(* CODESYS project oaksmodbuslibrary.library
   Title: oaksModbusLibrary
   Version: 1.1
   Placeholder: oaksModbusLibrary
   Company: Oaks AB

Project tree, tasks and I/O mapping:
  libraries: OaksLibrary, 1.1 (OaksAB); Tc2_BA, 3.3.9.0 (Beckhoff Automation GmbH); Tc2_ModbusSrv, 3.3.2.0 (Beckhoff Automation GmbH); Tc2_Standard, 3.3.3.0 (Beckhoff Automation GmbH); Tc2_System, 3.4.24.0 (Beckhoff Automation GmbH); Tc2_Utilities, 3.3.47.0 (Beckhoff Automation GmbH); Tc3_BA, 1.1.5.0 (Beckhoff Automation GmbH); Tc3_BA_Common, 2.1.4.0 (Beckhoff Automation GmbH); Tc3_Module, 3.3.21.0 (Beckhoff Automation GmbH)
  oaksModbusLibrary/
    [obsolete]/
      function block fbRCCC3DOCS [ST]
      function block fbSioxDamper [ST]
      function block fbWriteHoldingDoubleControlled [ST]
      function fHyst [ST]
    Belimo/
      Spjällställdon/
        function block fbBelimoLHVD3MOD [ST]
        function block fbBelimoUK24MOD [ST]
    Bitzer/
      function block fbBitzerSEi1 [ST]
    Calectro/
      function block fbCalair [ST]
      function block fbCalectroIoMb02 [ST]
    Daikin/
      function block fbDaikinRTDNET [ST]
    Danfoss/
      function block fbDanfossDGS_HFC [ST]
      function block fbDanfossEKE347 [ST]
    Datahantering/
      function F_INT_TO_WORD [ST]
      function F_WORD_TO_INT [ST]
      function block FB_SETPOINT_INT_MODBUS [ST]
      function block FB_SETPOINT_REAL_MODBUS [ST]
      function block fbDoubleControlledModbusHolding [ST]
      function block fbHoldingRWReadBackEEPROM_BOOL [ST]
      function block fbHoldingRWReadBackEEPROM_REAL [ST]
      function block fbReadGeneralModbusReg [ST]
      function block fbReadWriteCoilRegBool [ST]
      function block fbReadWriteHoldingReg [ST]
      function block fbReadWriteHoldingRegReal [ST]
      function fWordToReal [ST]
    DUTs/
      data type E_Modbus_Functions_Read
      data type ST_ModbusConfig
      data type ST_ModbusData
      data type ST_ModbusResultRegister
      data type ST_ModbusTCP
      data type U_WORD_INT
    EBM Papst/
      function block fbEbmPapst [ST]
    EcoGuard/
      function block fbEcocomTemperature [ST]
    Ej Testat/
    Elvaco/
      CME3100/
        Givare/
          function block fbElvacoTemperature [ST]
          function block fbElvacoTemperatureCo2 [ST]
          function block fbElvacoTemperatureHumidity [ST]
        Mätare/
          function block fbElvacoElectricMeter [ST]
          function block fbElvacoElectricMeterEnergy [ST]
          function block fbElvacoEnergyMeter [ST]
          function block fbElvacoWaterMeter [ST]
        function block fbElvacoGeneral [ST]
    Eveco/
      function block fbEveco [ST]: mSpeedEnableCheck
    Fidelix/
      FXIO (IO-kort)/
        Givarblock/
          function block fbFxIO_Sensor [ST]: mGT, mRaw
        Modulblock/
          function block fbFxIO_AI8 [ST]: mAI
          function block fbFxIO_AO8 [ST]
          function block fbFxIO_Combi36 [ST]
          function block fbFxIO_DI16 [ST]
          function block fbFxIO_DO8 [ST]
    Fläktwoods/
      Spjällställdon/
        function block fbFlaktwoods227PMMB [ST]
        function block fbFlaktwoods227VMMB [ST]
    Frico/
      function block fbFricoSirE [ST]: mBHyst
      function block fbFricoSirEOvride [ST]: mBHyst
    Grundfil/
      function block fbGrundfil [ST]
    Grundfos/
      function block fbGrundfosCIM [ST]
      function block fbGrundfosModbusMagna [ST]
    Gruner/
      Givare/
        function block fbGrunerGTVMDD3MB [ST]
      Spjällställdon/
        function block fbGruner227CMXXMB [ST]
    IMI hydronic/
      function block fbImiBrainCubeConnect [ST]
    Iv produkt/
      function block fbIvClimatixEnvistarIndication [ST]
      function block fbIvClimatixEnvistarOperationLevel [CFC]: mCommunicationAlarm, mIpadressString, mSpeedChoice
      function block fbIvSaphirOperationLevel [CFC]: mCommunicationAlarm, mIpadressString, mSpeedChoice
    IVT/
      function block fbIvtRego5200BorVarde [ST]
    Metz/
      DUT/
        data type E_MetzAIsensorConfig
        data type ST_MetzAI8config
        data type ST_MetzAI8Sensor
      Givare/
        function block fbMetzMR_AI8GeneralSensor [ST]
        function block fbMetzMR_AI8TempSensor [ST]
      function block fbMetzMR_AI8 [ST]: config
      function block fbMetzMR_AOP4 [ST]: mAnalogToRaw, mAnalogToRawFallback, mRawToAnalog
      function block fbMetzMR_DI10 [ST]
      function block fbMetzMR_DI4 [ST]
      function block fbMetzMR_DO4 [ST]: mAnalogToRaw, mAnalogToRawFallback, mRawToAnalog
      function block fbMetzMR_MULTI [ST]: config, mAnalogIn, mAnalogOut, mAnalogToRaw, mAnalogToRawFallback, mDigitalIn, mDigitalOut, mRawToAnalog
    Mitsubishi/
      function block fbMitsubishiATA_ATW [ST]
      function block fbMitsubishiHydroBox [ST]
    Nicotra Gebhardt/
      function block fbNicotraGebhardtRLM [ST]
    Produal/
      Givare/
        function block fbProdualHdhmCo2 [ST]
        function block fbProdualHdhmPirCo2 [ST]
        function block fbProdualHdhmTempCo2 [ST]
        function block fbProdualKLH [ST]
        function block fbProdualPEL2500Mx [ST]
      ProximaRIO/
        function block fbProximaCULH_RIO [ST]: mADConfig, mINConfig
        function block fbProximaRIO_Sensor [ST]: mDataIn
        data type ST_ProximaCULH_IO_Config
      Regulatorer/
        HLS44/
          function block fbProdualHLS44 [ST]
          function block fbProdualHLS44_IO [ST]
        function block fbProdualHdhmCo2Override [ST]
        function block fbProdualHdhmCo2PirOverride [ST]
    Regin/
      Givare/
        function block fbCthrc [ST]
        function block fbCtrc [ST]
      Regio midi/
        function block fbReginRCC [ST]
        function block fbReginRCC_CO2 [ST]
        function block fbReginRCC_Handst_Spjall [ST]
        function block fbReginRCC_Handst_Spjall_Co2 [ST]
    Schneider/
      function block fbAltivarATV600 [ST]
    Server-block/
      RTU/
        function block fbMbRtuSlaveCoilRegBool [ST]
        function block fbMbRtuSlaveHoldingRegInt [ST]
        function block fbMbRtuSlaveHoldingRegReal [ST]
        function block fbMbRtuSlaveHoldingRegUInt [ST]
        function block fbMbRtuSlaveStatusRegBool [ST]
      function block fbMbSlaveRegBool [ST]
      function block fbMbSlaveRegInt [ST]
      function block fbMbSlaveRegReal [ST]
      function block fbMbSlaveRegUInt [ST]
    Siemens/
      Spjäll/
        function block fbSiemensGDB1811EMO [ST]
    Siox/
      Via modul/
        function block fbSioxDamperDUOdirect [ST]
        function block fbSioxDamperUNOdirect [ST]
        function block fbSioxSxAcura [ST]
      Via SX-Access/
        function block fbSioxDamperDUO [ST]
        function block fbSioxDamperUNO [ST]
      function block fbSioxSxAcess [ST]
    Swegon/
      function block fbSwegonGoldCdOperationLevel [CFC]: mCommunicationAlarm, mIpadressString, mSpeedChoice
      function block fbSwegonGoldIndication [ST]
      function block fbSwegonGoldOperationLevel [CFC]: mCommunicationAlarm, mIpadressString, mSpeedChoice
      function block fbSwegonReact [ST]: mFlodesBalansering, mFlodesKompensering1, mFlodesKompensering10, mFlodesKompensering11, mFlodesKompensering12, mFlodesKompensering13, mFlodesKompensering14, mFlodesKompensering15, mFlodesKompensering2, mFlodesKompensering3, mFlodesKompensering4, mFlodesKompensering5, mFlodesKompensering6, mFlodesKompensering7, mFlodesKompensering8, mFlodesKompensering9, mOperationMode
      function block fbSwegonReactPx [ST]
      function block fbSwegonWiseMasterSlave [ST]
    Vacon/
      function block fbVaconFO_1 [ST]
    Wilo/
      function block fbWiloCif_If [ST]
    Xylem/
      function block fbXylemEcocircXLplus [ST]
      function block fbXylemHydrovarHVL [ST]
  ClassDiagram
  global variables GVL_ModbusRtuSlave
  global variables ModbusServer
*)

// oaksModbusLibrary/DUTs/E_Modbus_Functions_Read
{attribute 'qualified_only'}
{attribute 'strict'}
TYPE E_Modbus_Functions_Read :
(
	ReadCoils 			:= 1,
	ReadInputStatus 	:= 2,
	ReadHoldingRegister	:= 3,
	ReadInputRegister	:= 4
);
END_TYPE

// oaksModbusLibrary/DUTs/ST_ModbusConfig
TYPE ST_ModbusConfig :
STRUCT
	bEnable 		: BOOL; // IF TRUE, the slave is present and will be read from terminal. If FALSE no read are done and no update of values
	eMBFunction		: E_Modbus_Functions_Read; //MODBUS FUNCTION to use.
	nUnitId			: BYTE; // The MOdbus DeviceId of slave (1..247)
	nQuantity		: WORD :=1; // Quantity of registers or coils to be read out from slave (1..125 for holding/input registers, 1..2000 for coils)
	nMBAddr			: WORD; // The startaddress of the register or coil to be read out from slave
	tTimeBetwRead 	: TIME :=T#500MS; // Time before readout of the slave
END_STRUCT
END_TYPE

// oaksModbusLibrary/DUTs/ST_ModbusData
TYPE ST_ModbusData :
STRUCT
	aModbusData			: ARRAY [1..1000] OF WORD;
	aModbusGoodRead		: ARRAY [1..1000] OF BOOL;
	aModbusAddress		: ARRAY [1..1000] OF UINT;
	aModbusTimestamp	: ARRAY [1..1000] OF DT;
END_STRUCT
END_TYPE

// oaksModbusLibrary/DUTs/ST_ModbusResultRegister
TYPE ST_ModbusResultRegister :
STRUCT
	bEnable 		: BOOL; // IF TRUE, the slave is present and will be read from terminal. If false no read are done and no update of values
	eMBFunction		: E_Modbus_Functions_Read; //MODBUS FUNCTION that have been used
	nUnitId			: BYTE; // The MOdbus DeviceId of slave (1..247)
	nQuantity		: WORD; // Quantity of registers or coils to be read out from slave (1..125 for holding/input registers, 1..2000 for coils)
	nMBAddr			: WORD; // The startaddress of the register or coil to be read out from slave
	aRegisterArray	: ARRAY [1..125] OF WORD; // The telegram maximum length is 125 values of WORD.
	bReadSuccessful	: BOOL; // If the last read out from slave is without error then this value is TRUE, else FALSE
	DTLastRead		: TIMESTRUCT; // The date and time for the last reafout from slave (the values in aRegisterarray is from this date)
	stModbusError	: ST_ModbusErrorDiagnostics; // Error diagnostics from the last readout
	
END_STRUCT
END_TYPE

// oaksModbusLibrary/DUTs/ST_ModbusTCP
TYPE ST_ModbusTCP :
STRUCT
	sIPAddr : STRING := ''; //Ip-adress
	nTCPPort : UINT; //Modbus-TCP port
	iModbusLoop : INT :=1; //Modbusslinga
END_STRUCT
END_TYPE

// oaksModbusLibrary/DUTs/U_WORD_INT
TYPE U_WORD_INT :
UNION
	nWord	: WORD;
	nINT	: INT;
END_UNION
END_TYPE

// oaksModbusLibrary/Metz/DUT/E_MetzAIsensorConfig
{attribute 'qualified_only'}
{attribute 'strict'}
{attribute 'to_string'}
TYPE E_MetzAIsensorConfig :
(
Sensor_PT100 := 0,
Sensor_PT500 := 1,
Sensor_PT1000 := 2,
Sensor_NI1000_TK5000 := 3,
Sensor_NI1000_TK6180 := 4,
Sensor_BALCO_500 := 5,
Sensor_KTY81_110 := 6,
Sensor_KTY81_210 := 7,
Sensor_NTC_1k8 := 8,
Sensor_NTC_5k := 9,
Sensor_NTC_10k := 10,
Sensor_NTC_20k := 11,
Sensor_LM235 := 12,
Sensor_NTC_10k_CAREL := 13
);
END_TYPE

// oaksModbusLibrary/Metz/DUT/ST_MetzAI8config
TYPE ST_MetzAI8config :
STRUCT
	bResistance : BOOL :=FALSE; //0=0-10v, 1=Resistans
	sensorType : E_MetzAIsensorConfig := 2;  
END_STRUCT
END_TYPE

// oaksModbusLibrary/Metz/DUT/ST_MetzAI8Sensor
TYPE ST_MetzAI8Sensor :
STRUCT
	rRawValue : REAL := 0; //Rå-värde från IO-modul 
	bComError : BOOL := FALSE; //Kommunikationsfel från IO-modul
	sSensorConfig : STRING := ' '; 
END_STRUCT
END_TYPE

// oaksModbusLibrary/Produal/ProximaRIO/ST_ProximaCULH_IO_Config
TYPE ST_ProximaCULH_IO_Config :
STRUCT
	nInType 	: BYTE;
	nInRType	: BYTE; //0=Ohm, 1=DI
	nInDelay	: BYTE;
	
	nOutType	: BYTE; //0=0..10V, 1=PWM
	iOutPW		: INT;

	bError		: BOOL;	
END_STRUCT
END_TYPE

// GVL_ModbusRtuSlave
{attribute 'qualified_only'}
VAR_GLOBAL PERSISTENT
mb_Input    :  ARRAY [0..999] OF WORD;
mb_Output 	:  ARRAY [0..999] OF WORD;
mb_Memory	:  ARRAY [0..999] OF WORD;
END_VAR

// ModbusServer
{attribute 'qualified_only'}
VAR_GLOBAL
	mb_HoldingRegs 	:    ARRAY [0..999] OF WORD;
	mb_Coils	 	:    ARRAY [0..999] OF BOOL;
END_VAR

// oaksModbusLibrary/[obsolete]/fbRCCC3DOCS
//OAKS AB
//2020-03-17
//Funktionsblock för modbus-TCP, Regin RCC-C3DOCS rumsreglator (Endast som börvärdesomställare) bör ej användas för rumsstyrning.
// Specifikt för krokslätts fabriker.
{attribute 'obsolete' := 'Använd ersättningsblock. Detta block vidareutvecklas ej.'}
FUNCTION_BLOCK fbRCCC3DOCS
VAR_INPUT
	sIPAddr : STRING := ''; 
	nTCPPort : UINT := 502;
	nUnitID : UINT :=1;
	iModbusLoop : INT :=1; //Modbusslinga
	iMode : INT; //Driftläge 0=Off 1=Unoccupied, 2=Stand-by, 3=Occupied, 4=Bypass 
	bBlockDisplay : BOOL := TRUE;  //Blockering display
	iSetViewDisp : INT;//Visningsläge i display 0=Ärvärde, 1=Värmebörvärde, 2=Kylbörvärde, 3=Medelvärdet av värme och kylbörvärdet, 4=Endast börvärdesjusteringen, se modbuslista Adr 51
	iSetvalDisp : INT; //Visning av börvärde vid börvärdesjustering, se modbuslista Adr 52
	iBypassTime : INT; //Bypass-tid (min)
	rActSetpoint : REAL; //Aktuellt börvärde
	rActMaxSetpoint : REAL; //Max börvärdeförskjutning
	rActMinSetpoint : REAL; //Min börvärdeförskjutning
END_VAR

VAR_OUTPUT
	PV AT %M* : REAL;//Rumstemperatur~wp:[unit]°C[format]0.0[trendoptions]i:300
	PV1 AT %M* : INT;//Koldioxid~wp:[unit]ppm[format]0[trendoptions]i:300
	PV2 AT %M* : REAL;//Aktuell börvärdesförskjutning~wp:[unit]°C[format]0.0[trendoptions]i:300
	PV7 AT %M* : INT;//Modbus-ID~wp:[format]0
	PV8 AT %M* : INT;//Driftläge~wp:[format]0[trendoptions]i:300
	PV9 AT %M* : REAL;//Max lokal börvärdesförskutning~wp:[unit]°C[format]0.0[trendoptions]i:300
	PV10 AT %M* : REAL;//Min lokal börvärdesförskutning~wp:[unit]°C[format]0.0[trendoptions]i:300
	
	FAULT AT %M* : BOOL;//Kommunikationsfel~wp:
END_VAR

VAR
	//General
	offset : INT;
	rTemp : REAL;
	iTemp : INT;
	wTemp : WORD;
	bSekvensFlagga : BOOL;
	bBlockDisplayRead :  BOOL;
	
	//Read Coils
	FB_MBReadCoils_BlockDisp: FB_MBReadCoils;
	FB_MBWriteCoils_BlockDisp: FB_MBWriteCoils;
	
	//Read input registers
	FB_MBReadInputRegs_wArrInput1: FB_MBReadInputRegs;
	wArrInputRegs1 : ARRAY [1..12] OF WORD; //Input register function 4
		
	FB_MBReadInputRegs_wCo2: FB_MBReadInputRegs;		
	wCO2 : WORD; //Input register function 4
	
	//Read Holding	
	FB_MBReadRegs_Mode : FB_MBReadRegs;
	wModeRead : WORD; //Aktuellt driftläge 0=Off 1=Unoccupied, 2=Stand-by, 3=Occupied, 4=Bypass 

	FB_MBReadRegs_wArrHolding1 : FB_MBReadRegs;
	wArrHolding1 : ARRAY [51..60] OF WORD; //Holding
	wViewDispRead : WORD; //Visningsläge display, se modbus-lista
	wSetValDispRead : WORD; //Visningsläge börvärde, se modbus-lista
	wBypassTimeRead : WORD; //Tid i by-pass läge
		
	FB_MBReadRegs_wArrHolding2: FB_MBReadRegs;
	wArrHolding2 : ARRAY [61..80] OF WORD; //Holding
	wActSetpointRead : WORD; //Grundbörvärde kyla
	wActMaxSetpointRead : WORD; //Max förskjutning lokalt börvärde
	wActMinSetpointRead : WORD; //Min förskjutning lokalt börvärde
	wActOffsetRead : WORD; //Börvärdesjustering
	
	//Write Holding
	FB_MBWriteSingleReg_Mode : FB_MBWriteSingleReg;
	FB_MBWriteSingleReg_SetView : FB_MBWriteSingleReg;
	FB_MBWriteSingleReg_SetDisp : FB_MBWriteSingleReg;
	FB_MBWriteSingleReg_Bypasstime : FB_MBWriteSingleReg;
	FB_MBWriteSingleReg_Setpoint : FB_MBWriteSingleReg;
	FB_MBWriteSingleReg_MaxSetpoint : FB_MBWriteSingleReg;
	FB_MBWriteSingleReg_MinSetpoint : FB_MBWriteSingleReg;
	
	//Kommunikationsfel
	fbKommTof : tof; 
	fbKommTon : ton;
	
	FB_MBReadRegs_ArrHolding1: INT;
	bError: INT;
END_VAR

//General
	offset := -1;
//Sekvens	
	bSekvensFlagga := oaksGVL.aBModbusSekvens[iModbusLoop] = UINT_TO_INT(nUnitID);
//Modbus-ID
	PV7 :=  UINT_TO_INT(nUnitID);
///////////////		
//READ
///////////////			

//Read/Write Coils
	
	//Block display read
	FB_MBReadCoils_BlockDisp(
		sIPAddr:= sIpAddr, 
		nTCPPort:= INT_TO_UINT(nTCPPort), 
		nUnitID:= INT_TO_BYTE(nUnitID), 
		nQuantity:=1, 
		nMBAddr:= 21 + offset, 
		cbLength:= SIZEOF(bBlockDisplayRead), 
		pDestAddr:= ADR(bBlockDisplayRead), 
		bExecute:= bSekvensFlagga, 
		tTimeout:= T#3S, 
		bBusy=> , 
		bError=> , 
		nErrId=> , 
		cbRead=> );
				
		IF bBlockDisplay <> bBlockDisplayRead AND bSekvensFlagga THEN
			FB_MBWriteCoils_BlockDisp.bExecute := TRUE;
		ELSE
			FB_MBWriteCoils_BlockDisp.bExecute := FALSE;
		END_IF

	//Block display write	
	FB_MBWriteCoils_BlockDisp(
		sIPAddr:= sIpAddr, 
		nTCPPort:= INT_TO_UINT(nTCPPort), 
		nUnitID:= INT_TO_BYTE(nUnitID), 
		nQuantity:= 1, 
		nMBAddr:= 21 + offset, 
		cbLength:= SIZEOF(bBlockDisplay), 
		pSrcAddr:= ADR(bBlockDisplay), 
		bExecute:= , 
		tTimeout:= , 
		bBusy=> , 
		bError=> , 
		nErrId=> );	

		
//Read input registers function 4		

	//Read Array1
	FB_MBReadInputRegs_wArrInput1(
		sIPAddr:= sIpAddr, 
		nTCPPort:= INT_TO_UINT(nTCPPort), 
		nUnitID:= INT_TO_BYTE(nUnitID), 
		nQuantity:= 12, 
		nMBAddr:= 1 + offset, 
		cbLength:= SIZEOF(wArrInputRegs1), 
		pDestAddr:= ADR(wArrInputRegs1), 
		bExecute:= bSekvensFlagga, 
		tTimeout:= T#3S, 
		bBusy=> , 
		bError=> , 
		nErrId=> , 
		cbRead=> );
	
		//Values
		//wArrInputRegs1[1]; //1
		//wArrInputRegs1[2]; //2
		//wArrInputRegs1[3]; //3
		//wArrInputRegs1[4]; //4
		//wArrInputRegs1[5]; //5
		//wArrInputRegs1[6]; //6
		//wArrInputRegs1[7]); //7
		//wArrInputRegs1[8]; //8
		//wArrInputRegs1[9]; //9
		//wArrInputRegs1[10]; //10
		iTemp := WORD_TO_INT(wArrInputRegs1[11]); //11
		rTemp := INT_TO_REAL(iTemp); 
		PV := rTemp /10;
		//wArrInputRegs1[12]; //12
	
	//Read CO2		
	FB_MBReadInputRegs_wCo2(
		sIPAddr:= sIpAddr, 
		nTCPPort:= INT_TO_UINT(nTCPPort), 
		nUnitID:= INT_TO_BYTE(nUnitID), 
		nQuantity:= 1, 
		nMBAddr:= 32 + offset, 
		cbLength:= SIZEOF(wCO2), 
		pDestAddr:= ADR(wCO2), 
		bExecute:= bSekvensFlagga, 
		tTimeout:= T#3S, 
		bBusy=> , 
		bError=> , 
		nErrId=> , 
		cbRead=> );
	
		PV1 := WORD_TO_INT(wCO2); //32

//Read Holding registers function 3		

	//Read Mode
	FB_MBReadRegs_Mode(
		sIPAddr:= sIpAddr, 
		nTCPPort:= INT_TO_UINT(nTCPPort), 
		nUnitID:= INT_TO_BYTE(nUnitID), 
		nQuantity:= 1, 
		nMBAddr:= 14+offset, 
		cbLength:= SIZEOF(wModeRead), 
		pDestAddr:= ADR(wModeRead), 
		bExecute:= bSekvensFlagga, 
		tTimeout:= T#3S, 
		bBusy=> , 
		bError=> , 
		nErrId=> , 
		cbRead=> );

		PV8 := WORD_TO_INT(wModeRead);
		
	//Read Array1	
	FB_MBReadRegs_wArrHolding1(
		sIPAddr:= sIpAddr, 
		nTCPPort:= INT_TO_UINT(nTCPPort), 
		nUnitID:= INT_TO_BYTE(nUnitID), 
		nQuantity:= 10, 
		nMBAddr:= 51+offset, 
		cbLength:= SIZEOF(wArrHolding1), 
		pDestAddr:= ADR(wArrHolding1), 
		bExecute:= bSekvensFlagga, 
		tTimeout:= T#3S, 
		bBusy=> , 
		bError=> , 
		nErrId=> , 
		cbRead=> );
		
		//Values
		wViewDispRead := wArrHolding1[51]; //51
		wSetValDispRead := wArrHolding1[52]; //52
		//wArrHolding1[53]; //53
		//wArrHolding1[54]; //54
		//wArrHolding1[55]; //55
		wBypassTimeRead := wArrHolding1[56]; //56
		//wArrHolding1[57]; //57
		//wArrHolding1[58]; //58
		//wArrHolding1[59]; //59
		//wArrHolding1[60]; //60

	//Read Array2	
	FB_MBReadRegs_wArrHolding2(
		sIPAddr:= sIpAddr, 
		nTCPPort:= INT_TO_UINT(nTCPPort), 
		nUnitID:= INT_TO_BYTE(nUnitID), 
		nQuantity:= 20, 
		nMBAddr:= 61+offset, 
		cbLength:= SIZEOF(wArrHolding2), 
		pDestAddr:= ADR(wArrHolding2), 
		bExecute:= bSekvensFlagga, 
		tTimeout:= T#3S, 
		bBusy=> , 
		bError=> , 
		nErrId=> , 
		cbRead=> );
		
		//Values
		//wArrHolding2[61]; //61
		//wArrHolding2[62]; //62
		//wArrHolding2[63]; //63
		//wArrHolding2[64]; //64
		//wArrHolding2[65]; //65
		//wArrHolding2[66]; //66
		//wArrHolding2[67]; //67
		//wArrHolding2[68]; //68
		wActSetpointRead := (wArrHolding2[69]); //69
		//wArrHolding2[70]; //70
		//wArrHolding2[71]; //71
		//wArrHolding2[72]; //72
		//wArrHolding2[73]; //73
		
		wActMaxSetpointRead := (wArrHolding2[74]); //74
		iTemp := WORD_TO_INT(wActMaxSetpointRead);		
		PV9 := iTemp / 10;
		
		wActMinSetpointRead := (wArrHolding2[75]); //75
		iTemp := WORD_TO_INT(wActMinSetpointRead);	
		PV10 := iTemp /10;
		
		wActOffsetRead := (wArrHolding2[76]); //76
		iTemp := WORD_TO_INT(wActOffsetRead);
		PV2 := iTemp / 10;
		
		//wArrHolding2[77]; //77
		//wArrHolding2[78]; //78
		//wArrHolding2[79]; //79
		//wArrHolding2[80]; //80

//Write Holding registers

	//Write mode
	wTemp := INT_TO_WORD(iMode);
	
	IF (wModeRead) <> wTemp AND bSekvensFlagga THEN
		FB_MBWriteSingleReg_Mode.bExecute := TRUE;
	ELSE
		FB_MBWriteSingleReg_Mode.bExecute := FALSE;
	END_IF

	FB_MBWriteSingleReg_Mode(
		sIPAddr:= sIpAddr , 
		nTCPPort:= INT_TO_UINT(nTCPPort), 
		nUnitID:= INT_TO_BYTE(nUnitID), 
		nMBAddr:= 14 + offset, 
		nValue:= wTemp, 
		bExecute:= , 
		tTimeout:= T#5S , 
		bBusy=> , 
		bError=> , 
		nErrId=> );
	
	//Write Viewmode
	wTemp := INT_TO_WORD(iSetViewDisp);
	
	IF wViewDispRead <> wTemp AND bSekvensFlagga THEN
		FB_MBWriteSingleReg_SetView.bExecute := TRUE;
	ELSE
		FB_MBWriteSingleReg_SetView.bExecute := FALSE;
	END_IF

	FB_MBWriteSingleReg_SetView(
		sIPAddr:= sIpAddr , 
		nTCPPort:= INT_TO_UINT(nTCPPort), 
		nUnitID:= INT_TO_BYTE(nUnitID), 
		nMBAddr:= 51 + offset, 
		nValue:= wTemp, 
		bExecute:= , 
		tTimeout:= T#5S , 
		bBusy=> , 
		bError=> , 
		nErrId=> );
		
	//Write DisplaySetpoint Mode
	wTemp := INT_TO_WORD(iSetvalDisp);
	
	IF wSetValDispRead <> wTemp AND bSekvensFlagga THEN
		FB_MBWriteSingleReg_SetDisp.bExecute := TRUE;
	ELSE
		FB_MBWriteSingleReg_SetDisp.bExecute := FALSE;
	END_IF

	FB_MBWriteSingleReg_SetDisp(
		sIPAddr:= sIpAddr , 
		nTCPPort:= INT_TO_UINT(nTCPPort), 
		nUnitID:= INT_TO_BYTE(nUnitID), 
		nMBAddr:= 52 + offset, 
		nValue:= wTemp, 
		bExecute:= , 
		tTimeout:= T#5S , 
		bBusy=> , 
		bError=> , 
		nErrId=> );

	//Write Bypass-time
	wTemp := INT_TO_WORD(iBypassTime);
	
	IF wBypassTimeRead <> wTemp AND bSekvensFlagga THEN
		FB_MBWriteSingleReg_Bypasstime.bExecute := TRUE;
	ELSE
		FB_MBWriteSingleReg_Bypasstime.bExecute := FALSE;
	END_IF

	FB_MBWriteSingleReg_Bypasstime(
		sIPAddr:= sIpAddr , 
		nTCPPort:= INT_TO_UINT(nTCPPort), 
		nUnitID:= INT_TO_BYTE(nUnitID), 
		nMBAddr:= 56 + offset, 
		nValue:= wTemp, 
		bExecute:= , 
		tTimeout:= T#5S , 
		bBusy=> , 
		bError=> , 
		nErrId=> );

	//Setpoint
	iTemp := REAL_TO_INT(rActSetpoint * 10);
	wTemp := INT_TO_WORD(iTemp);
	
	IF wActSetpointRead <> wTemp AND bSekvensFlagga THEN
		FB_MBWriteSingleReg_Setpoint.bExecute := TRUE;
	ELSE
		FB_MBWriteSingleReg_Setpoint.bExecute := FALSE;
	END_IF

	FB_MBWriteSingleReg_Setpoint(
		sIPAddr:= sIpAddr , 
		nTCPPort:= INT_TO_UINT(nTCPPort), 
		nUnitID:= INT_TO_BYTE(nUnitID), 
		nMBAddr:= 69 + offset, 
		nValue:= wTemp, 
		bExecute:= , 
		tTimeout:= T#5S , 
		bBusy=> , 
		bError=> , 
		nErrId=> );
	
	//Max Setpoint
	iTemp := REAL_TO_INT(rActMaxSetpoint * 10);
	wTemp := INT_TO_WORD(iTemp);
	
	IF wActMaxSetpointRead <> wTemp AND bSekvensFlagga THEN
		FB_MBWriteSingleReg_MaxSetpoint.bExecute := TRUE;
	ELSE
		FB_MBWriteSingleReg_MaxSetpoint.bExecute := FALSE;
	END_IF

	FB_MBWriteSingleReg_MaxSetpoint(
		sIPAddr:= sIpAddr , 
		nTCPPort:= INT_TO_UINT(nTCPPort), 
		nUnitID:= INT_TO_BYTE(nUnitID), 
		nMBAddr:= 74 + offset, 
		nValue:= wTemp, 
		bExecute:= , 
		tTimeout:= T#5S , 
		bBusy=> , 
		bError=> , 
		nErrId=> );	
		
	//Min Setpoint
	iTemp := REAL_TO_INT(rActMinSetpoint * 10);
	wTemp := INT_TO_WORD(iTemp);
	
	IF wActMinSetpointRead <> wTemp AND bSekvensFlagga THEN
		FB_MBWriteSingleReg_MinSetpoint.bExecute := TRUE;
	ELSE
		FB_MBWriteSingleReg_MinSetpoint.bExecute := FALSE;
	END_IF

	FB_MBWriteSingleReg_MinSetpoint(
		sIPAddr:= sIpAddr , 
		nTCPPort:= INT_TO_UINT(nTCPPort), 
		nUnitID:= INT_TO_BYTE(nUnitID), 
		nMBAddr:= 75 + offset, 
		nValue:= wTemp, 
		bExecute:= , 
		tTimeout:= T#5S , 
		bBusy=> , 
		bError=> , 
		nErrId=> );	

//Communication error
	fbKommTof(IN:=FB_MBReadCoils_BlockDisp.bError OR
	FB_MBWriteCoils_BlockDisp.bError OR		
	FB_MBReadInputRegs_wArrInput1.bError OR
	FB_MBReadInputRegs_wCo2.bError OR	
	FB_MBReadRegs_Mode.bError OR
	FB_MBReadRegs_wArrHolding1.bError OR
	FB_MBReadRegs_wArrHolding2.bError OR
	FB_MBWriteSingleReg_Mode.bError OR
	FB_MBWriteSingleReg_SetView.bError OR
	FB_MBWriteSingleReg_SetDisp.bError OR
	FB_MBWriteSingleReg_Bypasstime.bError OR
	FB_MBWriteSingleReg_Setpoint.bError OR
	FB_MBWriteSingleReg_MaxSetpoint.bError OR
	FB_MBWriteSingleReg_MinSetpoint.bError,
	PT:=T#20S , Q=> , ET=> );
	fbKommTon(IN:=fbKommTof.Q , PT:=T#20M , Q=> , ET=> );
	FAULT :=fbKommTon.Q;

//Write busy	
	oaksgvl.aBModbusBusyFlagga[iModbusLoop,nUnitID] := FB_MBReadCoils_BlockDisp.bBusy OR
	FB_MBWriteCoils_BlockDisp.bBusy OR		
	FB_MBReadInputRegs_wArrInput1.bBusy OR
	FB_MBReadInputRegs_wCo2.bBusy OR	
	FB_MBReadRegs_Mode.bBusy OR
	FB_MBReadRegs_wArrHolding1.bBusy OR
	FB_MBReadRegs_wArrHolding2.bBusy OR
	FB_MBWriteSingleReg_Mode.bBusy OR
	FB_MBWriteSingleReg_SetView.bBusy OR
	FB_MBWriteSingleReg_SetDisp.bBusy OR
	FB_MBWriteSingleReg_Bypasstime.bBusy OR
	FB_MBWriteSingleReg_Setpoint.bBusy OR
	FB_MBWriteSingleReg_MaxSetpoint.bBusy OR
	FB_MBWriteSingleReg_MinSetpoint.bBusy;

END_FUNCTION_BLOCK

// oaksModbusLibrary/[obsolete]/fbSioxDamper
{attribute 'obsolete' := 'Använd ersättningsblock. Detta block vidareutvecklas ej.'}
FUNCTION_BLOCK fbSioxDamper

VAR_INPUT
	sIPAddr: STRING(15) := '192.168.1.32';
	iPort: UINT := 502;
	iUnitID : BYTE := 60;
	iAdress : WORD := 257;
END_VAR
VAR_OUTPUT
	FAULT AT %M*  : BOOL; //Kommunikationsfel Siox~wp:[trendoptions]i:300
	V AT %M*  : BOOL; //Standby bit (1=Standby)~wp:[trendoptions]i:300
	PV5 AT %M*  : BOOL; //Motionskörning~wp:[trendoptions]i:300
	AL AT %M*  : BOOL; //Övertemperatur (NTC)~wp:[trendoptions]i:300  
	DAMPER1_AL  AT %M*  : BOOL; //Driftfel spjäll 1~wp:[trendoptions]i:300  
	DAMPER1_V0  AT %M*  : BOOL; //Stängtindikering spjäll 1~wp:[trendoptions]i:300
	DAMPER1_V1  AT %M*  : BOOL; //Öppetindikering spjäll 1~wp:[trendoptions]i:300
	DAMPER2_AL  AT %M*  : BOOL; //Driftfel spjäll 2~wp:[trendoptions]i:300
	DAMPER2_V0  AT %M*  : BOOL; //Stängtindikering spjäll 2~wp:[trendoptions]i:300
	DAMPER2_V1  AT %M*  : BOOL; //Öppetindikering spjäll 2~wp:[trendoptions]i:300
	GX_AL  AT %M*  : BOOL; //Utlöst rökdetektor~wp:[trendoptions]i:300
	GX_AL1  AT %M*  : BOOL;  //Servicelarm rökdetektor~wp:[trendoptions]i:300
	GX_AL2  AT %M*  : BOOL; //Slingfel~wp:[trendoptions]i:300
	GX_V  AT %M*  : BOOL; //Rökdetektor I drift~wp:[trendoptions]i:300
	PV8 AT %M* : STRING;//Modbus konfiguering~wp:
END_VAR
VAR

	wInternalWord : WORD;
	fbKommTof: Tof;
	fbKommTon: Ton;
	FB_MBReadRegs01: FB_MBReadRegs;
	fbtoggle1 : fbToggle;
	
		sIP: STRING(255);
	sPort: STRING(255);
	sModbusID: STRING(255);
	sModbusLoop: STRING(255);
	sTemp : STRING(255);
END_VAR

//Modbus konfiguering
	sIP := CONCAT (SIPAddr, '');
	sPort := CONCAT ('<br>Port: ', UINT_TO_STRING(iPort)); 								
	sModbusID := CONCAT('<br>ID: ', UINT_TO_STRING(iUnitID));
	sModbusLoop := CONCAT('<br>Adress: ', INT_TO_STRING(iAdress));	

	sTemp := sIP;
	sTemp := CONCAT(sTemp, sPort);
	sTemp := CONCAT(sTemp, sModbusID);
	sTemp := CONCAT(sTemp, sModbusLoop);
	
	PV8 := sTemp;

fbtoggle1(bStart:=TRUE , bOutput=>,tTimeOn := T#1S,tTimeOff := T#1S );

	fbKommTof(IN:=FB_MBReadRegs01.bError , PT:=T#3S , Q=> , ET=> );
	fbKommTon(IN:=fbKommTof.Q , PT:=T#15M , Q=> , ET=> );
	FAULT :=fbKommTon.Q;

FB_MBReadRegs01(
	sIPAddr:= sIPAddr, 
	nTCPPort:= iPort, 
	nUnitID:= iUnitID, 
	nQuantity:= 1, 
	nMBAddr:= iAdress, 
	cbLength:= SIZEOF(wInternalWord), 
	pDestAddr:=ADR(wInternalWord) , 
	bExecute:=fbtoggle1.bOutput , 
	tTimeout:= , 
	bBusy=> , 
	bError=> , 
	nErrId=> , 
	cbRead=> );
	
	V := wInternalWord.0;
	PV5 := wInternalWord.4;
	AL :=  wInternalWord.7;
	DAMPER1_AL := wInternalWord.3;
	DAMPER1_V0 := wInternalWord.8;
	DAMPER1_V1 := wInternalWord.9;
	DAMPER2_AL := wInternalWord.5;
	DAMPER2_V0 := wInternalWord.10;
	DAMPER2_V1 := wInternalWord.11;
	GX_AL := wInternalWord.13;
	GX_AL1 := wInternalWord.14;
	GX_AL2 := wInternalWord.15;
	GX_V := wInternalWord.12;
(*

SIOX_GROUP10_PV4	SIOX	40267.0	UINT	0	0	0	0			Standby bit (1=Standby)	 	0
SIOX_GROUP10_PV5	SIOX	40267.4	UINT	0	0	0	0			Motionskörning	 	0
SIOX_GROUP11_AL	SIOX	40268.7	UINT	0	0	0	0			Övertemperatur (NTC)	  	0
SIOX_GROUP11_DAMPER1_AL	SIOX	40268.3	UINT	0	0	0	0			Driftfel spjäll 1	  	0
SIOX_GROUP11_DAMPER1_V0	SIOX	40268.8	UINT	0	0	0	0			Stängtindikering spjäll 1	 	1
SIOX_GROUP11_DAMPER1_V1	SIOX	40268.9	UINT	0	0	0	0			Öppetindikering spjäll 1	 	0
SIOX_GROUP11_DAMPER2_AL	SIOX	40268.5	UINT	0	0	0	0			Driftfel spjäll 2	  	0
SIOX_GROUP11_DAMPER2_V0	SIOX	40268.1	UINT	0	0	0	0			Stängtindikering spjäll 2	 	1
SIOX_GROUP11_DAMPER2_V1	SIOX	40268.11	UINT	0	0	0	0			Öppetindikering spjäll 2	 	0
SIOX_GROUP11_GX_AL	SIOX	40268.13	UINT	0	0	0	0			Utlöst rökdetektor	  	0
SIOX_GROUP11_GX_AL1	SIOX	40268.14	UINT	0	0	0	0			Servicelarm rökdetektor	  	0
SIOX_GROUP11_GX_AL2	SIOX	40268.15	UINT	0	0	0	0			Slingfel	  	0
SIOX_GROUP11_GX_V	SIOX	40268.12	UINT	0	0	0	0			Rökdetektor I drift		(0)
*)

END_FUNCTION_BLOCK

// oaksModbusLibrary/[obsolete]/fbWriteHoldingDoubleControlled
{attribute 'obsolete' := 'Använd ersättningsblock. Detta block vidareutvecklas ej.'}
FUNCTION_BLOCK fbWriteHoldingDoubleControlled
VAR_IN_OUT
	wWriteInput : WORD;
END_VAR
VAR_INPUT
	sIPAddr : STRING;
	nTCPPort : UINT;
	nUnitID : BYTE;
	nMBAddr : UINT;
	bEnable : BOOL;
END_VAR
VAR_OUTPUT
	bBusy : BOOL;
	bError : BOOL;
	nErrId : UDINT;
END_VAR
VAR
	fbHoldingRead : FB_MBReadRegs;
	fbHoldingWrite: FB_MBWriteSingleReg;
	wReadWord : WORD;
	fbCheckReg : FbDoubleControlledVariableWord;
	bEnableWrite : BOOL ;
	wValueToWrite : WORD;
	fbToggle01 : fbToggle;
	wTemp : WORD;
END_VAR

	fbHoldingRead(
	sIPAddr:=sIPAddr , 
	nTCPPort:=nTCPPort , 
	nUnitID:= nUnitID, 
	nQuantity:=1 , 
	nMBAddr:=nMBAddr , 
	cbLength:= SIZEOF(wReadWord), 
	pDestAddr:=ADR(wReadWord) , 
	bExecute:=bEnable , 
	tTimeout:=T#5S , 
	bBusy=>bBusy , 
	bError=> bError, 
	nErrId=>nErrId , 
	cbRead=> );
	
	//test
// Kolla om vi ska skriva till register med hjälp av en avancerad algoritm för dubbelsidig paramterförändring 

wTemp := wReadWord;
fbCheckReg(wVariableInPLC:=wWriteInput, wVariableInModbusUnit:=wTemp);
IF wWriteInput <> wReadWord THEN
	wValueToWrite := INT_TO_WORD(wWriteInput);
	bEnableWrite := TRUE;
ELSE
	bEnableWrite := FALSE;
END_IF
	
fbToggle01(bStart:=bEnableWrite , tTimeOn:=T#1S , tTimeOff:=T#1S , bOutput=> );
	
	
	fbHoldingWrite(
	sIPAddr:= sIpAddr, 
	nTCPPort:= nTCPPort, 
	nUnitID:= nUnitID, 
	nMBAddr:= nMBAddr, 
	nValue:= wValueToWrite, 
	bExecute:= fbToggle01.bOutput, 
	tTimeout:=T#5S , 
	bBusy=> , 
	bError=> , 
	nErrId=> );

END_FUNCTION_BLOCK

// oaksModbusLibrary/[obsolete]/fHyst
FUNCTION fHyst : bool
VAR_INPUT
	rProcessValue : REAL;
	rSetPoint : REAL; 
	rDevLimit : REAL;
END_VAR
VAR
END_VAR

	IF rProcessValue > (rSetPoint + rDevLimit)  THEN
		fHyst := TRUE;
	ELSIF rProcessValue < (rSetPoint - rDevLimit)  THEN
		fHyst := TRUE;
	ELSE	
		fHyst := FALSE;
	END_IF;

END_FUNCTION

// oaksModbusLibrary/Belimo/Spjällställdon/fbBelimoLHVD3MOD
//OAKS AB
//2020-03-17
//Funktionsblock för modbus-TCP, Belimo LHV/LMV-D3-MOD (linjärt/vridande spjällställdon). Mätning ställs att visa m3/h i spjäll. Omräkning till l/s sker i funktionsblock.
FUNCTION_BLOCK fbBelimoLHVD3MOD
VAR_INPUT
	sIPAddr : STRING := ''; 
	nTCPPort : UINT;
	nUnitID : UINT :=1;
	iModbusLoop : INT :=1; //Modbusslinga
	rSetpoint : REAL; //Börvärde
	iMode : INT; //Överstyrning spjäll-läge 0: None 1: Open 2: Close 3: Min 4: Mid 5: MAX
	SP1 AT %M* : REAL;//Min-flöde~wp:[unit]%[format]0[trendoptions]i:300
	SP2 AT %M* : REAL;//Max-flöde~wp:[unit]%[format]0[trendoptions]i:300	
		
END_VAR
VAR_OUTPUT
	
	PV1 AT %M* : REAL;//Volym~wp:[unit]l/s[format]0[trendoptions]i:300
	PV5 AT %M* : UINT;//Spjäll-läge 0: None 1: Open 2: Close 3: Min 4: Mid 5: MAX~wp:[format]0[trendoptions]i:14400, t:1
	PV6 AT %M* : UINT;//Nominellt volym flöde~wp:[unit]m3/h[format]0[trendoptions]i:14400, t:1
	PV7 AT %M* : REAL;//Inställt min-flöde~wp:[unit]l/s[format]0[trendoptions]i:14400, t:1
	PV8 AT %M* : REAL;//Inställt max-flöde~wp:[unit]l/s[format]0[trendoptions]i:14400, t:1
	PV9 AT %M* : REAL;//Inställt min-flöde~wp:[unit]%[format]0[trendoptions]i:14400, t:1
	PV10 AT %M* : REAL;//Inställt max-flöde~wp:[unit]%[format]0[trendoptions]i:14400, t:1
	PV11 AT %M* : STRING;//Modbus konfigurering~wp:
	CSP AT %M* : REAL;//Uträknat börvärde~wp:[unit]l/s[format]0[trendoptions]i:300
	OP AT %M* : REAL;//Relativ position~wp:[unit]%[format]0[trendoptions]i:300	
	FAULT AT %M* : BOOL;//Kommunikationsfel~wp:
	
END_VAR
VAR
	offset : WORD :=0;
	offsetExtends : WORD :=0;
	rTemp : REAL;
	iTemp : UINT;
	wTemp : WORD;
	bSekvensFlagga : BOOL;
	
	FB_MBReadRegs_ArrHolding1: FB_MBReadRegs;
	wArrHolding1 : ARRAY [0..12] OF WORD; //Holding
	wActSetpoint : WORD; //Börvärde 0
	wModeOut : WORD; //Överstyrning 1 
	wRelPos : WORD; //Relativ position 4
	wAbsVolume : WORD; //Volym 7

	FB_MBReadRegs_ArrHolding2 : FB_MBReadRegs;
	wArrHolding2 : ARRAY [99..118] OF WORD; //Holding	
	wAlarm : WORD; //Fel 104
	wVmin : WORD; //Min setpoint 105
	wVmax : WORD; //Max setpoint 106
	wNomVolFlow : WORD; //Nominellt volym flöde m3/h
	
	FB_MBWriteSingleReg_Setpoint : FB_MBWriteSingleReg; 
	FB_MBWriteSingleReg_Mode : FB_MBWriteSingleReg; 
	
	//Skrivning
	fbWriteHoldingDoubleControlledMin: fbDoubleControlledModbusHolding;
	fbWriteHoldingDoubleControlledMax: fbDoubleControlledModbusHolding;
	
	//Kommunikationsfel
	fbKommTof : tof; 
	fbKommTon : ton;
	
	fb_CSP : Tc3_BA.FB_BA_Chrct02;	
		
	sIP: STRING(255);
	sPort: STRING(255);
	sModbusID: STRING(255);
	sModbusLoop: STRING(255);
	sTemp : STRING(255);
	
END_VAR

VAR_IN_OUT

END_VAR

//General
	offset := 0 + offsetExtends;
//Sekvens	
	bSekvensFlagga := oaksGVL.aBModbusSekvens[iModbusLoop] = UINT_TO_INT(nUnitID);
//Modbus konfiguering
	sIP := CONCAT (SIPAddr, '');
	sPort := CONCAT ('<br>Port: ', UINT_TO_STRING(nTCPPort)); 								
	sModbusID := CONCAT('<br>ID: ', UINT_TO_STRING(nUnitID));
	sModbusLoop := CONCAT('<br>Loop: ', INT_TO_STRING(iModbusLoop));	

	sTemp := sIP;
	sTemp := CONCAT(sTemp, sPort);
	sTemp := CONCAT(sTemp, sModbusID);
	sTemp := CONCAT(sTemp, sModbusLoop);
	
	PV11 := sTemp;
 
///////////////		
//READ
///////////////		
	
	//Read Holding 0-12
	FB_MBReadRegs_ArrHolding1(
	sIPAddr:= sIpAddr, 
	nTCPPort:= INT_TO_UINT(nTCPPort), 
	nUnitID:= INT_TO_BYTE(nUnitID), 
	nQuantity:= 12, 
	nMBAddr:= 0 + offset, 
	cbLength:= SIZEOF(wArrHolding1), 
	pDestAddr:= ADR(wArrHolding1), 
	bExecute:= bSekvensFlagga, 
	tTimeout:= T#3S, 
	bBusy=> , 
	bError=> , 
	nErrId=> , 
	cbRead=> );
	
		//Values
		wActSetpoint := wArrHolding1[0]; //0
		wModeOut := wArrHolding1[1]; //1
		//wArrHolding1[2]; //2
		//wArrHolding1[3]; //3
		wRelPos := wArrHolding1[4]; //4
		//wArrHolding1[5]; //5
		//wArrHolding1[6]; //6
		wAbsVolume := wArrHolding1[7]; //7
		//wArrHolding1[8]; //8
		//wArrHolding1[9]; //9
		//wArrHolding1[10]; //10
		//wArrHolding1[11]; //11
		//wArrHolding1[12]; //12
						
		//Absolute Volume flow
		//Converter from m2 to l/s
		iTemp := WORD_TO_UINT(wAbsVolume);
		rTemp := UINT_TO_REAL(iTemp);
		PV1 := rTemp / 3.6;
	
		//Relative Position
		iTemp := WORD_TO_UINT(wRelPos);
		rTemp := UINT_TO_REAL(iTemp);
		OP := rTemp / 100;
		
		//Actual damper-mode
		PV5 := WORD_TO_UINT(wModeOut);
						
	//Read Holding 99-118
	FB_MBReadRegs_ArrHolding2(
	sIPAddr:= sIpAddr, 
	nTCPPort:= INT_TO_UINT(nTCPPort), 
	nUnitID:= INT_TO_BYTE(nUnitID), 
	nQuantity:= 20, 
	nMBAddr:= 99 + offset, 
	cbLength:= SIZEOF(wArrHolding2), 
	pDestAddr:= ADR(wArrHolding2), 
	bExecute:= bSekvensFlagga, 
	tTimeout:= T#3S, 
	bBusy=> , 
	bError=> , 
	nErrId=> , 
	cbRead=> );
	
		//Tilldela värden
		//wArrHolding2[99]; //99
		//wArrHolding2[100]; //100
		//wArrHolding2[101]; //101
		//wArrHolding2[102]; //102
		//wArrHolding2[103]; //103
		wAlarm := wArrHolding2[104]; //104
		wVmin := wArrHolding2[105]; //105
		wVmax := wArrHolding2[106]; //106
		//wArrHolding2[107]; //107
		//wArrHolding2[108]; //108
		//wArrHolding2[109]; //109
		wNomVolFlow := wArrHolding2[110]; //110
		//wArrHolding2[111]; //111
		//wArrHolding2[112]; //112
		//wArrHolding2[113]; //113
		//wArrHolding2[114]; //114
		//wArrHolding2[115]; //115
		//wArrHolding2[116]; //116
		//wArrHolding2[117]; //117
		//wArrHolding2[118]; //118
			
		//Nominal Volume flow (m2/h)
		PV6 := wNomVolFlow;
					
		//Setpoint min-flow (Calculation l/s + %)
		iTemp := WORD_TO_UINT(wVmin);
		rTemp := UINT_TO_REAL(iTemp);
		
		PV7 :=  (rTemp /10000) * (wNomVolFlow / 3.6) ;
		PV9 :=  (rTemp /100);		
				
		//Setpoint max-flow (Calculation l/s + %)
		iTemp := WORD_TO_UINT(wVmax);
		rTemp := UINT_TO_REAL(iTemp);		
		PV8 := (rTemp /10000) * (wNomVolFlow / 3.6);
		PV10 := (rTemp /100);
		
		//Calculated setpoint
		CSP := (WORD_TO_REAL(wNomVolFlow) / 3.6) * (WORD_TO_REAL(wActSetpoint) / 10000);
		
		//Calculated setpoint
		fb_CSP(
			rX:= WORD_TO_REAL(wActSetpoint) / 100, 
			rX01:= 0, 
			rX02:= 100, 
			rY01:= PV7, 
			rY02:= PV8, 
			bLmt:= TRUE, 
			rY=> CSP, 
			bErr=> , 
			sErrDescr=> );
					
		
///////////////		
//WRITE
///////////////	
				
//Setpoint
	rTemp := LIMIT (0, rSetpoint, 100);
	wTemp := frealtoword(rTemp, 100);
	
	IF wTemp <> wActSetpoint AND bSekvensFlagga THEN
		FB_MBWriteSingleReg_Setpoint.bExecute := TRUE;
	ELSE
		FB_MBWriteSingleReg_Setpoint.bExecute := FALSE;
	END_IF
	
	//Write Setpoint
	FB_MBWriteSingleReg_Setpoint(
	sIPAddr:= sIpAddr, 
	nTCPPort:= INT_TO_UINT(nTCPPort), 
	nUnitID:= INT_TO_BYTE(nUnitID), 
	nMBAddr:= 0 + offset, 
	nValue:= wTemp, 
	bExecute:= , 
	tTimeout:= T#3S, 
	bBusy=> , 
	bError=> , 
	nErrId=> );
	
//Override

	iTemp := INT_TO_WORD(iMode);	
	
	IF wModeOut <> iTemp AND bSekvensFlagga THEN 
		FB_MBWriteSingleReg_Mode.bExecute := TRUE;
	ELSE 
		FB_MBWriteSingleReg_Mode.bExecute := FALSE;
	END_IF
	
	//Write Mode
	FB_MBWriteSingleReg_Mode(
	sIPAddr:= sIpAddr, 
	nTCPPort:= INT_TO_UINT(nTCPPort), 
	nUnitID:= INT_TO_BYTE(nUnitID), 
	nMBAddr:= 1 + offset, 
	nValue:= UINT_TO_WORD(iTemp), 
	bExecute:= , 
	tTimeout:= T#3S, 
	bBusy=> , 
	bError=> , 
	nErrId=> );

//Read/write

//Min
	fbWriteHoldingDoubleControlledMin(
	sIPAddr:= sIPAddr, 
	nTCPPort:= nTCPPort, 
	nUnitID:= UINT_TO_BYTE(nUnitID) , 
	nMBAddr:= 105+offset, 
	bExecute:= bSekvensFlagga, 
	rScale:= 100, 
	rWrite:= SP1, 
	bBusy=> , 
	bError=> );
//Max		
	fbWriteHoldingDoubleControlledMax(
	sIPAddr:= sIPAddr, 
	nTCPPort:= nTCPPort, 
	nUnitID:= UINT_TO_BYTE(nUnitID) , 
	nMBAddr:= 106+offset, 
	bExecute:= bSekvensFlagga, 
	rScale:= 100, 
	rWrite:= SP2, 
	bBusy=> , 
	bError=> );
	

	
//Communication error
	fbKommTof(IN:=FB_MBReadRegs_ArrHolding1.bError , PT:=T#20S , Q=> , ET=> );
	fbKommTon(IN:=fbKommTof.Q , PT:=T#20M , Q=> , ET=> );
	FAULT :=fbKommTon.Q;
		
//Write busy	
	oaksgvl.aBModbusBusyFlagga[iModbusLoop,nUnitID] := FB_MBReadRegs_Arrholding1.bBusy OR FB_MBReadRegs_Arrholding2.bBusy OR FB_MBWriteSingleReg_Setpoint.bBusy OR FB_MBWriteSingleReg_Mode.bBusy;

END_FUNCTION_BLOCK

// oaksModbusLibrary/Datahantering/fbDoubleControlledModbusHolding
FUNCTION_BLOCK fbDoubleControlledModbusHolding
VAR_INPUT
	sIPAddr : STRING := ''; 
	nTCPPort : UINT := 502;
	nUnitID : BYTE :=1;
	nMBAddr : WORD := 1;
	bExecute : BOOL;
	rScale : REAL;
	tTimeout : TIME := T#10S;
	tStartDelay : TIME := T#20MS;
END_VAR
VAR_IN_OUT
	rWrite : REAL; // Variabel att skriva
END_VAR 
VAR_OUTPUT
	bBusy : BOOL;
	bError : BOOL;
END_VAR
VAR
	fbStartDelayTon : TON;
	FB_SETPOINT_REAL_MODBUS01 : FB_SETPOINT_REAL_MODBUS;
	fbHoldingWrite: FB_MBWriteSingleReg;
	fbHoldingRead : FB_MBReadRegs;
	wValueToWrite : WORD;
		
	nTempCompLow		: REAL; 	//Calectro CalAir HoldingRegister 18
	nTempCompLowWord		: WORD; 	//Calectro CalAir HoldingRegister 18
	
	fbReadTrig : r_trig; 
END_VAR

	fbStartDelayTon(IN:=bExecute , PT:=tStartDelay , Q=> , ET=> );

	fbHoldingRead(
	sIPAddr:= sIPAddr, 
	nTCPPort:= nTCPPort, 
	nUnitID:= nUnitID, 
	nMBAddr:= nMBAddr, 
	nQuantity:=1 , 
	cbLength:= SIZEOF(nTempCompLowWord), 
	pDestAddr:=ADR(nTempCompLowWord) , 
	bExecute:=fbStartDelayTon.Q , 
	tTimeout:=tTimeout , 
	bBusy=> , 
	bError=> , 
	nErrId=> , 
	cbRead=> );
	
	nTempCompLow := INT_TO_REAL(F_WORD_TO_INT(nTempCompLowWord));
	
	fbReadTrig(CLK:= NOT fbHoldingRead.bBusy AND NOT fbHoldingRead.bError);
	
	FB_SETPOINT_REAL_MODBUS01(
	bPrioritySlave:= TRUE, 
	bSuccessModbusSlave:=fbReadTrig.Q , 
	fActSetpointSlave:= nTempCompLow, 
	bValidPLCMaster:= TRUE, 
	tMaxTime:= T#60S, 
	fScale := rScale,
	fSetpointPLCMaster:= rWrite, 
	fSetpointValid=> , 
	nSetpointToSlave=>wValueToWrite , 
	bSetpointUpdateSlave=> );
	
	fbHoldingWrite(
	sIPAddr:= sIPAddr, 
	nTCPPort:= nTCPPort, 
	nUnitID:= nUnitID, 
	nMBAddr:= nMBAddr, 
	nValue:= wValueToWrite, 
	bExecute:= FB_SETPOINT_REAL_MODBUS01.bSetpointUpdateSlave, 
	tTimeout:=tTimeout , 
	bBusy=> , 
	bError=> , 
	nErrId=> );
	
	bBusy := fbHoldingRead.bBusy OR fbHoldingWrite.bBusy;
	bError := fbHoldingRead.bError OR fbHoldingWrite.bError;

END_FUNCTION_BLOCK

// oaksModbusLibrary/Datahantering/F_WORD_TO_INT
FUNCTION F_WORD_TO_INT : INT
VAR_INPUT
	nWordInput	: WORD;	
END_VAR

VAR
	uWordToInt	: U_WORD_INT;
END_VAR

uWordToInt.nWord:= nWordInput;
F_WORD_TO_INT:= uWordToInt.nINT;

END_FUNCTION

// oaksModbusLibrary/Datahantering/FB_SETPOINT_REAL_MODBUS
FUNCTION_BLOCK FB_SETPOINT_REAL_MODBUS
VAR_INPUT
	bPrioritySlave			: BOOL	:=TRUE;
	bSuccessModbusSlave		: BOOL;
	fActSetpointSlave		: REAL;
	bValidPLCMaster			: BOOL;
	tMaxTime				: TIME	:=T#30S;
	fScale					: REAL	:=1;
				 					
END_VAR

VAR_IN_OUT
	fSetpointPLCMaster		: REAL;
END_VAR

VAR_OUTPUT
	fSetpointValid			: REAL;
	nSetpointToSlave		: WORD;
	bSetpointUpdateSlave	: BOOL;
END_VAR

VAR
	fMemorySetpoint			: REAL;
	nSeq					: INT;
	fbTimerMax				: TON;
END_VAR

fbTimerMax();

IF fScale = 0 THEN fScale := 1; END_IF

CASE nSeq OF
	0: (* Start up case first time, after power failure and max time elapsed *)
		IF bPrioritySlave AND bSuccessModbusSlave THEN
			fSetpointPLCMaster:= fActSetpointSlave;
			fMemorySetpoint:= fActSetpointSlave;
			fSetpointValid:= fActSetpointSlave;
			nSetpointToSlave:=F_INT_TO_WORD(REAL_TO_INT(fSetpointValid*fScale));
			bSetpointUpdateSlave:= FALSE;
			nSeq :=10;
		END_IF

		
	10: (* Control of setpoint change *)
		IF bSuccessModbusSlave AND fMemorySetpoint <> (fActSetpointSlave / fScale) THEN
			nSeq :=20;
		ELSIF bSuccessModbusSlave AND fMemorySetpoint <> fSetpointPLCMaster  THEN
			nSeq :=30;
		END_IF

		
	20: (* Slave changed setpoint *)
			fSetpointPLCMaster:= fActSetpointSlave /fScale;
			fMemorySetpoint:= fActSetpointSlave / fScale;
			fSetpointValid:= fActSetpointSlave / fScale;
			nSetpointToSlave:=F_INT_TO_WORD(REAL_TO_INT(fSetpointValid*fScale));
			bSetpointUpdateSlave:= FALSE;
			nSeq :=10;

	
	30: (* PLC Master changed setpoint *)
			fMemorySetpoint:= fSetpointPLCMaster;
			fSetpointValid:= fSetpointPLCMaster;
			nSetpointToSlave:=F_INT_TO_WORD(REAL_TO_INT(fSetpointValid*fScale));
			bSetpointUpdateSlave:= TRUE;
			nSeq :=31;

			
	31: (* Waiting for slave to change setpoint *)
			fbTimerMax(IN:=bSetpointUpdateSlave , PT:= tMaxTime, Q=> , ET=> );
		IF fMemorySetpoint = fActSetpointSlave THEN
			bSetpointUpdateSlave:= FALSE;
			fbTimerMax.IN := bSetpointUpdateSlave;
			nSeq :=10;
		ELSIF fbTimerMax.Q THEN
			bSetpointUpdateSlave:=FALSE;
			fbTimerMax.IN := bSetpointUpdateSlave;
			fbTimerMax();
			nSeq:=0;
		END_IF;

	
END_CASE

END_FUNCTION_BLOCK

// oaksModbusLibrary/Datahantering/F_INT_TO_WORD
FUNCTION F_INT_TO_WORD : WORD
VAR_INPUT
	nIntInput	: INT;
END_VAR

VAR
	uWordToInt	: U_WORD_INT;
END_VAR

uWordToInt.nINT:= nIntInput;
F_INT_TO_WORD:= uWordToInt.nWord;

END_FUNCTION

// oaksModbusLibrary/Belimo/Spjällställdon/fbBelimoUK24MOD
//OAKS AB
//2020-03-17
//Funktionsblock för modbus-TCP, Belimo UK24-MOD (linjärt/vridande spjällställdon). Mätning ställs att visa m3/h i spjäll. Omräkning till l/s sker i funktionsblock.
//Funktion är samma som LHVDMOD men konmmunikation sker mot en modbus-gateway som kommunicerar med underliggande spjäll. Register för förskjutna med en fast offeset om 20/40/60 osv. 
FUNCTION_BLOCK fbBelimoUK24MOD
VAR_INPUT
	sIPAddr : STRING := ''; 
	nTCPPort : UINT;
	nUnitID : UINT :=1;
	iModbusLoop : INT :=1; //Modbusslinga
	rSetpoint : REAL; //Börvärde
	iMode : INT; //Överstyrning spjäll-läge 0: None 1: Open 2: Close 3: Min 4: Mid 5: MAX
	SP1 AT %M* : REAL;//Min-flöde~wp:[unit]%[format]0[trendoptions]i:300
	SP2 AT %M* : REAL;//Max-flöde~wp:[unit]%[format]0[trendoptions]i:300
	iOffsetMpBus : INT; //Offset MP-Bus	
		
END_VAR
VAR_OUTPUT
	
	PV1 AT %M* : REAL;//Volym~wp:[unit]l/s[format]0[trendoptions]i:300
	PV5 AT %M* : UINT;//Spjäll-läge 0: None 1: Open 2: Close 3: Min 4: Mid 5: MAX~wp:[format]0[trendoptions]i:14400, t:1
	PV6 AT %M* : UINT;//Nominellt volym flöde~wp:[unit]m3/h[format]0[trendoptions]i:14400, t:1
	PV7 AT %M* : REAL;//Inställt min-flöde~wp:[unit]l/s[format]0[trendoptions]i:14400, t:1
	PV8 AT %M* : REAL;//Inställt max-flöde~wp:[unit]l/s[format]0[trendoptions]i:14400, t:1
	PV9 AT %M* : REAL;//Inställt min-flöde~wp:[unit]%[format]0[trendoptions]i:14400, t:1
	PV10 AT %M* : REAL;//Inställt max-flöde~wp:[unit]%[format]0[trendoptions]i:14400, t:1
	PV11 AT %M* : STRING;//Modbus konfigurering~wp:
	CSP AT %M* : REAL;//Uträknat börvärde~wp:[unit]l/s[format]0[trendoptions]i:300
	OP AT %M* : REAL;//Relativ position~wp:[unit]%[format]0[trendoptions]i:300	
	FAULT AT %M* : BOOL;//Kommunikationsfel~wp:
	
END_VAR
VAR
	offset : WORD :=0;
	rTemp : REAL;
	iTemp : UINT;
	wTemp : WORD;
	bSekvensFlagga : BOOL;
	
	FB_MBReadRegs_ArrHolding1: FB_MBReadRegs;
	wArrHolding1 : ARRAY [0..17] OF WORD; //Holding
	wActSetpoint : WORD; //Börvärde 0
	wModeOut : WORD; //Överstyrning 1 
	wRelPos : WORD; //Relativ position 4
	wAbsVolume : WORD; //Volym 7

	wAlarm : WORD; //Fel 104
	wVmin : WORD; //Min setpoint 105
	wVmax : WORD; //Max setpoint 106
	wNomVolFlow : WORD; //Nominellt volym flöde m2/h
	
	FB_MBWriteSingleReg_Setpoint : FB_MBWriteSingleReg; 
	FB_MBWriteSingleReg_Mode : FB_MBWriteSingleReg; 
	
	//Skrivning
	fbWriteHoldingDoubleControlledMin: fbDoubleControlledModbusHolding;
	fbWriteHoldingDoubleControlledMax: fbDoubleControlledModbusHolding;
	
	//Kommunikationsfel
	fbKommTof : tof; 
	fbKommTon : ton;
	
	fb_CSP : Tc3_BA.FB_BA_Chrct02;	
		
	sIP: STRING(255);
	sPort: STRING(255);
	sModbusID: STRING(255);
	sModbusLoop: STRING(255);
	sTemp : STRING(255);
	
END_VAR

VAR_IN_OUT

END_VAR

//General
	offset := 0 + INT_TO_WORD(iOffsetMpBus);
//Sekvens	
	bSekvensFlagga := oaksGVL.aBModbusSekvens[iModbusLoop] = UINT_TO_INT(nUnitID);
//Modbus konfiguering
	sIP := CONCAT (SIPAddr, '');
	sPort := CONCAT ('<br>Port: ', UINT_TO_STRING(nTCPPort)); 								
	sModbusID := CONCAT('<br>ID: ', UINT_TO_STRING(nUnitID));
	sModbusLoop := CONCAT('<br>Loop: ', INT_TO_STRING(iModbusLoop));	

	sTemp := sIP;
	sTemp := CONCAT(sTemp, sPort);
	sTemp := CONCAT(sTemp, sModbusID);
	sTemp := CONCAT(sTemp, sModbusLoop);
	
	PV11 := sTemp;
 
///////////////		
//READ
///////////////		
	
	//Read Holding 0-17
	FB_MBReadRegs_ArrHolding1(
	sIPAddr:= sIpAddr, 
	nTCPPort:= INT_TO_UINT(nTCPPort), 
	nUnitID:= INT_TO_BYTE(nUnitID), 
	nQuantity:= 17, 
	nMBAddr:= 0 + offset, 
	cbLength:= SIZEOF(wArrHolding1), 
	pDestAddr:= ADR(wArrHolding1), 
	bExecute:= bSekvensFlagga, 
	tTimeout:= T#3S, 
	bBusy=> , 
	bError=> , 
	nErrId=> , 
	cbRead=> );
	
		//Values
		wActSetpoint := wArrHolding1[0]; //0
		wModeOut := wArrHolding1[1]; //1
		//wArrHolding1[2]; //2
		wRelPos := wArrHolding1[3]; //3
		// wArrHolding1[4]; //4
		wAlarm := wArrHolding1[5]; //5
		//wArrHolding1[6]; //7
		//wArrHolding1[7]; //7
		//wArrHolding1[8]; //8
		//wArrHolding1[9]; //9
		//wArrHolding1[10]; //10
		//wArrHolding1[11]; //11
		//wArrHolding1[12]; //12
		wVmin := wArrHolding1[13]; //13
		wVmax := wArrHolding1[14]; //14
		wAbsVolume  := wArrHolding1[15]; //15
		wNomVolFlow := wArrHolding1[16]; //16		
		//wArrHolding1[17]; //17
		
								
		//Absolute Volume flow
		//Converter from m2 to l/s
		iTemp := WORD_TO_UINT(wAbsVolume);
		rTemp := UINT_TO_REAL(iTemp);
		PV1 := rTemp / 3.6;
	
		//Relative Position
		iTemp := WORD_TO_UINT(wRelPos);
		rTemp := UINT_TO_REAL(iTemp);
		OP := rTemp / 100;
		
		//Actual damper-mode
		PV5 := WORD_TO_UINT(wModeOut);
			
		//Nominal Volume flow (m2/h)
		PV6 := wNomVolFlow;
					
		//Setpoint min-flow (Calculation l/s + %)
		iTemp := WORD_TO_UINT(wVmin);
		rTemp := UINT_TO_REAL(iTemp);
		
		PV7 :=  (rTemp /10000) * (wNomVolFlow / 3.6) ;
		PV9 :=  (rTemp /100);		
				
		//Setpoint max-flow (Calculation l/s + %)
		iTemp := WORD_TO_UINT(wVmax);
		rTemp := UINT_TO_REAL(iTemp);		
		PV8 := (rTemp /10000) * (wNomVolFlow / 3.6);
		PV10 := (rTemp /100);
		
		//Calculated setpoint
		CSP := (WORD_TO_REAL(wNomVolFlow) / 3.6) * (WORD_TO_REAL(wActSetpoint) / 10000);
		
		//Calculated setpoint
		fb_CSP(
			rX:= WORD_TO_REAL(wActSetpoint) / 100, 
			rX01:= 0, 
			rX02:= 100, 
			rY01:= PV7, 
			rY02:= PV8, 
			bLmt:= TRUE, 
			rY=> CSP, 
			bErr=> , 
			sErrDescr=> );
					
		
///////////////		
//WRITE
///////////////	
				
//Setpoint
	rTemp := LIMIT (0, rSetpoint, 100);
	wTemp := frealtoword(rTemp, 100);
	
	IF iTemp <> wActSetpoint AND bSekvensFlagga THEN
		FB_MBWriteSingleReg_Setpoint.bExecute := TRUE;
	ELSE
		FB_MBWriteSingleReg_Setpoint.bExecute := FALSE;
	END_IF
	
	//Write Setpoint
	FB_MBWriteSingleReg_Setpoint(
	sIPAddr:= sIpAddr, 
	nTCPPort:= INT_TO_UINT(nTCPPort), 
	nUnitID:= INT_TO_BYTE(nUnitID), 
	nMBAddr:= 0 + offset, 
	nValue:= wTemp, 
	bExecute:= , 
	tTimeout:= T#3S, 
	bBusy=> , 
	bError=> , 
	nErrId=> );
	
//Override

	iTemp := INT_TO_WORD(iMode);	
	
	IF wModeOut <> iTemp AND bSekvensFlagga THEN 
		FB_MBWriteSingleReg_Mode.bExecute := TRUE;
	ELSE 
		FB_MBWriteSingleReg_Mode.bExecute := FALSE;
	END_IF
	
	//Write Mode
	FB_MBWriteSingleReg_Mode(
	sIPAddr:= sIpAddr, 
	nTCPPort:= INT_TO_UINT(nTCPPort), 
	nUnitID:= INT_TO_BYTE(nUnitID), 
	nMBAddr:= 1 + offset, 
	nValue:= UINT_TO_WORD(iTemp), 
	bExecute:= , 
	tTimeout:= T#3S, 
	bBusy=> , 
	bError=> , 
	nErrId=> );

//Read/write

//Min
	fbWriteHoldingDoubleControlledMin(
	sIPAddr:= sIPAddr, 
	nTCPPort:= nTCPPort, 
	nUnitID:= UINT_TO_BYTE(nUnitID) , 
	nMBAddr:= 13+offset,
	bExecute:= bSekvensFlagga, 
	rScale:= 100, 
	rWrite:=SP1 , 
	bBusy=> , 
	bError=> );
//Max
	fbWriteHoldingDoubleControlledMax(
	sIPAddr:= sIPAddr, 
	nTCPPort:= nTCPPort, 
	nUnitID:= UINT_TO_BYTE(nUnitID) , 
	nMBAddr:= 14+offset, 
	bExecute:= bSekvensFlagga, 
	rScale:=100 , 
	rWrite:= SP2, 
	bBusy=> , 
	bError=> );
	
//Communication error
	fbKommTof(IN:=FB_MBReadRegs_ArrHolding1.bError , PT:=T#20S , Q=> , ET=> );
	fbKommTon(IN:=fbKommTof.Q , PT:=T#20M , Q=> , ET=> );
	FAULT :=fbKommTon.Q;
		
//Write busy	
	oaksgvl.aBModbusBusyFlagga[iModbusLoop,nUnitID] := FB_MBReadRegs_Arrholding1.bBusy OR FB_MBWriteSingleReg_Setpoint.bBusy OR FB_MBWriteSingleReg_Mode.bBusy;

END_FUNCTION_BLOCK

// oaksModbusLibrary/Bitzer/fbBitzerSEi1
//Funktionsblock för kommunikation mot säkerhetsmodul Bitzer SE-i1 (via ModbusTCP-gateway). Skriv larmreset, läsning av div. värden. IO-enheter ej som WP-tagg.
//Robert H Oaks AB 
//22-03-22

//V 1.0	Testad

//OBS! Ej anpassad för Modbus-sekvens i oaks-standard, bör åtgärdas!!

(*



HR 110 Serial Control Word

IR 103 Status Word
IR 11104 If locked, ICP is
IR 11201 Code of highest alarm
IR 11202 Code of second highest alarm
...
IR 11205 Code of 5th rank alarm
IR 12001 Suction Pressure
IR 12002 Discharge Pressure
IR 12003 Evaporating Temperature (SST)
IR 12004 Condensing Temperature (SDT)
IR 12010 Discharge temperature
IR 12011 AUX temperature
*)



FUNCTION_BLOCK fbBitzerSEi1
VAR_INPUT
	sIPAddr 		: STRING; 			//Ip-adress till ModbusTCP-gateway
	nMBTCPPort		: UINT := 502;		//ModbusTCP-port
	nUnitID			: UINT := 1;		//Enhetsadress
	tInterval		: TIME := T#3S;		//Kommunikationsintervall
	tTimeout		: TIME := T#2.5S;	//Timeout
	CMD AT %M*		: BOOL;				//Larmreset ~wp: 
END_VAR

VAR_OUTPUT
	AL1		AT %M*		: BOOL;				//Varning säk.modul kompressor~wp:[alarmoptions]p:2
	V1		AT %M*		: BOOL;				//Kompressor i drift~wp:
	AL2		AT %M*		: BOOL;				//Kritisk varning säk.modul kompressor (risk för stopp)~wp:[alarmoptions]p:1,d:25
	V2		AT %M*		: BOOL;				//Kvittering behövs~wp:
	PV1 	AT %M*		: STRING :='';		//Nödvändig kvitteringsnivå~wp:[trendoptions]i:14400, t:1
	PV2		AT %M*		: UINT;				//Larmkod nivå 1 (se larmdok.)~wp:[trendoptions]i:14400, t:1
	PV3		AT %M*		: UINT;				//Larmkod nivå 2~wp:[trendoptions]i:14400, t:1
	PV4		AT %M*		: UINT;				//Larmkod nivå 3~wp:[trendoptions]i:14400, t:1
	PV5		AT %M*		: UINT;				//Larmkod nivå 4~wp:[trendoptions]i:14400, t:1
	PV6		AT %M*		: UINT;				//Larmkod nivå 5~wp:[trendoptions]i:14400, t:1
	AL8		AT %M*		: BOOL;				//Kommunikationsfel säkerhetsmodul kompressor~wp:[alarmoptions]p:2
		
	rPsuc		: REAL;		//Förångningstryck 				bar 	0.00
	rPdis		: REAL;		//Kondenseringstryck 			bar 	0.00
	rSatTempSuc	: REAL;		//Förångningstemp (beräknad)	°C		0.00
	rSatTempDis	: REAL;		//Kondenseringstemp (beräknad)	°C		0.00
	rTdis		: REAL;		//Hetgastemp (beräknad)			°C		0.00
	rTaux		: REAL;		//Temp AUX (beräknad)			°C		0.00		OBS t ex Suggas!
	nResLvlReq	: UINT;		//Nödvändig kvitteringsnivå index
	bOilFault	: BOOL;		//Indikering låg oljenivå
	rThermistor	: REAL;		//Motorskyddstermistor			Ohm		0
	
END_VAR

VAR
	bRun			: BOOL;	
	fbRunTON		: TON;
	fbRunTRIG		: R_TRIG;
	
	iCaseCMD		: INT;
	fbWriteTON		: TON;
	
	fbRHR110		: FB_MBReadRegs;
	fbWHR110		: FB_MBWriteSingleReg;
	
	fbRIR103		: FB_MBReadRegs;
	fbRIR11104		: FB_MBReadRegs;
	fbRIR11105		: FB_MBReadRegs;
	fbRIR11201_05	: FB_MBReadRegs;
	fbRIR12001_04	: FB_MBReadRegs;
	fbRIR12010_11	: FB_MBReadRegs;
	fbRIR12025		: FB_MBReadRegs;
	fbRIR13001		: FB_MBReadRegs;
	
	wRHR110			: WORD;
	wRIR103			: WORD;
	wRIR11104		: WORD;
	wRIR11105		: WORD;
	awRIR11201_05	: ARRAY[0..4] OF WORD;
	awRIR12001_04	: ARRAY[0..3] OF WORD;
	awRIR12010_11	: ARRAY[0..1] OF WORD;
	wRIR12025		: WORD;
	wRIR13001		: WORD;
	
	fbErrorTOF		: TOF;
	fbErrorTON		: TON;
	
END_VAR

fbRunTON(IN := NOT bRun, PT := tInterval);
fbRunTRIG(CLK := fbRunTON.Q, Q => bRun);


//HR 110 Serial Control Word		Endast larmreset. Läs in ord, då larmreset sätts från Webport skrivs ord tillbaks lika läsning med bit 2 & 10 hög, 
//									sedan med bit 2 & 10 låg igen	
fbRHR110.sIPAddr	:= sIPAddr;
fbRHR110.nTCPPort	:= nMBTCPPort;
fbRHR110.nUnitID 	:= UINT_TO_BYTE(nUnitID); 
fbRHR110.nQuantity	:= 1;
fbRHR110.tTimeout 	:= tTimeout;   
fbRHR110.nMBAddr 	:= 110;
fbRHR110.cbLength	:= SIZEOF(wRHR110);
fbRHR110.pDestAddr	:= ADR(wRHR110);

fbWHR110.sIPAddr	:= sIPAddr;
fbWHR110.nTCPPort	:= nMBTCPPort;
fbWHR110.nUnitID 	:= UINT_TO_BYTE(nUnitID); 
fbWHR110.tTimeout 	:= tTimeout;   
fbWHR110.nMBAddr 	:= 110;
fbWHR110.nValue		:= wRHR110;

IF CMD THEN				//Om larmreset

	fbRHR110.bExecute := FALSE;
	fbWHR110.bExecute := FALSE;
	
	CASE iCaseCMD OF
		0:				//Steg 0, läs in hela ordet och gå till steg 1
		fbRHR110.bExecute := TRUE;
		iCaseCMD := 1;
		
		1:				//Steg 1, när läsblocket ej är busy eller har felflagga, sätt bit 10 (serial control enable), vänta och gå sedan till steg 2
		fbWriteTON(IN := TRUE, PT := T#1S);
		
		IF NOT (fbRHR110.bBusy OR fbRHR110.bError) THEN
			
			wRHR110.10 	:= TRUE;
			
			fbWHR110.bExecute := TRUE;
				
		END_IF
		
		IF fbWriteTON.Q THEN
			fbWriteTON(IN := FALSE);
			fbWHR110.bExecute := FALSE;
			iCaseCMD := 2;
		END_IF
		
		2:				//Steg 2, när skrivblocket ej är busy eller har felflagga, sätt bit 7 (alarm reset), vänta och gå sedan till steg 3
		fbWriteTON(IN := TRUE, PT := T#1S);
		
		IF NOT (fbRHR110.bBusy OR fbRHR110.bError) THEN
			
			wRHR110.7 	:= TRUE;
			
			fbWHR110.bExecute := TRUE;
				
		END_IF
		
		IF fbWriteTON.Q THEN
			fbWriteTON(IN := FALSE);
			fbWHR110.bExecute := FALSE;
			iCaseCMD := 3;
		END_IF
		
		3:				//Steg 3, när skrivblocket ej är busy eller har felflagga, återställ bit 7 & 10 och skriv ordet, vänta och sedan återställ CMD och gå tbx till steg 0
		fbWriteTON(IN := TRUE, PT := T#1S);
		IF NOT (fbWHR110.bBusy OR fbWHR110.bError) THEN
			
			wRHR110.7 	:= FALSE;
			wRHR110.10 	:= FALSE;
			
			fbWHR110.bExecute := TRUE;
				
		END_IF
		
		IF fbWriteTON.Q THEN
			fbWriteTON(IN := FALSE);
			iCaseCMD := 0;
			CMD := FALSE;
		END_IF
		
	END_CASE
	
	fbRHR110();
	fbWHR110();

ELSE
	
	fbRHR110(bExecute := FALSE);
	fbWHR110(bExecute := FALSE);	
	
END_IF;



	
//IR 103 Status Word	
fbRIR103(sIPAddr := sIPAddr, nTCPPort := nMBTCPPort, nUnitID := UINT_TO_BYTE(nUnitID), nQuantity := 1, bExecute := bRun, tTimeout := tTimeout,   
	nMBAddr 	:= 103,
	cbLength	:= SIZEOF(wRIR103),
	pDestAddr	:= ADR(wRIR103));
	AL1		:= wRIR103.7;
	V1		:= wRIR103.11;
	AL2		:= wRIR103.13;
	
	
//IR 11104 If locked, ICP is (återställning behövs)	
fbRIR11104(sIPAddr := sIPAddr, nTCPPort := nMBTCPPort, nUnitID := UINT_TO_BYTE(nUnitID), nQuantity := 1, bExecute := bRun, tTimeout := tTimeout,   
	nMBAddr 	:= 11104,
	cbLength	:= SIZEOF(wRIR11104),
	pDestAddr	:= ADR(wRIR11104));
	V2	:= wRIR11104 > 0;
	
//IR 11105 Reset level required (vilken typ av återställning behövs)	
fbRIR11105(sIPAddr := sIPAddr, nTCPPort := nMBTCPPort, nUnitID := UINT_TO_BYTE(nUnitID), nQuantity := 1, bExecute := bRun, tTimeout := tTimeout,   
	nMBAddr 	:= 11105,
	cbLength	:= SIZEOF(wRIR11105),
	pDestAddr	:= ADR(wRIR11105));
	nResLvlReq	:= wRIR11105;
	
IF fbRIR11105.bError THEN
	PV1 := 'Offline';
ELSE	
	CASE wRIR11105 OF 
		0:
		PV1	:= 'Ingen (ej trippad)';
		1:
		PV1	:= 'Ingen (auto)';
		2:
		PV1	:= 'Ingen (auto fördröjd)';
		3:
		PV1	:= 'Via operatörspanel';
		4:
		PV1	:= 'Via omstart (knapp på AS)';
	END_CASE;
END_IF;
	
//IR 11201..05 Code of highest alarm..5th alarm	Läs ut larmkod för dom 5 allvarligaste larmerna (fallande ordning). Slå ut annan data i resp. ord med SHL/SHR
fbRIR11201_05(sIPAddr := sIPAddr, nTCPPort := nMBTCPPort, nUnitID := UINT_TO_BYTE(nUnitID), bExecute := bRun, tTimeout := tTimeout, 
	nQuantity 	:= 5,  
	nMBAddr 	:= 11201,
	cbLength	:= SIZEOF(awRIR11201_05),
	pDestAddr	:= ADR(awRIR11201_05));
	PV2		:= SHR(SHL(awRIR11201_05[0], 6), 6);
	PV3		:= SHR(SHL(awRIR11201_05[1], 6), 6);
	PV4		:= SHR(SHL(awRIR11201_05[2], 6), 6);
	PV5		:= SHR(SHL(awRIR11201_05[3], 6), 6);
	PV6		:= SHR(SHL(awRIR11201_05[4], 6), 6);
	
//IR 12001..04 	Avläsning givare
fbRIR12001_04(sIPAddr := sIPAddr, nTCPPort := nMBTCPPort, nUnitID := UINT_TO_BYTE(nUnitID), bExecute := bRun, tTimeout := tTimeout, 
	nQuantity 	:= 4,  
	nMBAddr 	:= 12001,
	cbLength	:= SIZEOF(awRIR12001_04),
	pDestAddr	:= ADR(awRIR12001_04));
	rPsuc		:= INT_TO_REAL(WORD_TO_INT(awRIR12001_04[0]));	//kPa
	rPdis		:= INT_TO_REAL(WORD_TO_INT(awRIR12001_04[1]));	//kPa
	rSatTempSuc	:= INT_TO_REAL(WORD_TO_INT(awRIR12001_04[2])) / 10;
	rSatTempDis	:= INT_TO_REAL(WORD_TO_INT(awRIR12001_04[3])) / 10; 
	
//IR 12010..11 	Avläsning givare
fbRIR12010_11(sIPAddr := sIPAddr, nTCPPort := nMBTCPPort, nUnitID := UINT_TO_BYTE(nUnitID), bExecute := bRun, tTimeout := tTimeout, 
	nQuantity 	:= 2,  
	nMBAddr 	:= 12010,
	cbLength	:= SIZEOF(awRIR12010_11),
	pDestAddr	:= ADR(awRIR12010_11));
	rTdis		:= INT_TO_REAL(WORD_TO_INT(awRIR12010_11[0])) / 10;
	rTaux		:= INT_TO_REAL(WORD_TO_INT(awRIR12010_11[1])) / 10;
	
//IR 12025 Oil Sensor 1	
fbRIR12025(sIPAddr := sIPAddr, nTCPPort := nMBTCPPort, nUnitID := UINT_TO_BYTE(nUnitID), nQuantity := 1, bExecute := bRun, tTimeout := tTimeout,   
	nMBAddr 	:= 12025,
	cbLength	:= SIZEOF(wRIR12025),
	pDestAddr	:= ADR(wRIR12025));
	bOilFault	:= wRIR12025 > 0;
	
//IR 13001 Motor overheat thermistor	
fbRIR13001(sIPAddr := sIPAddr, nTCPPort := nMBTCPPort, nUnitID := UINT_TO_BYTE(nUnitID), nQuantity := 1, bExecute := bRun, tTimeout := tTimeout,   
	nMBAddr 	:= 13001,
	cbLength	:= SIZEOF(wRIR13001),
	pDestAddr	:= ADR(wRIR13001));
	rThermistor	:= wRIR13001;
	
//Kom.fel modbus
fbErrorTOF(IN := fbRIR12010_11.bError, PT := T#5S);
fbErrorTON(IN := fbErrorTOF.Q, PT := T#120S, Q => AL8);

END_FUNCTION_BLOCK

// oaksModbusLibrary/Calectro/fbCalair
//OAKS AB
//2020-05-12
//Grundfil för modbusblock
FUNCTION_BLOCK fbCalair
VAR_INPUT
	sIPAddr : STRING := ''; 
	nTCPPort : UINT;
	nUnitID : UINT :=1;
	iModbusLoop : INT :=1; //Modbusslinga
	rSetpoint : REAL; // Börvärde (Pa)		
END_VAR
VAR_OUTPUT
	OP AT %M* : REAL; //Utsignal~wp:[unit]%[format]0[trendoptions]i:300
	PV AT %M* : REAL; //Aktuellt tryck~wp:[unit]Pa[format]0[trendoptions]i:300
	PV1 AT %M* : REAL; //Temperatur~wp:[unit]°C[format]0.0[trendoptions]i:300
	CSP AT %M* : REAL; //Aktuellt börvärde tryck~wp:[unit]Pa[format]0[trendoptions]i:300
	AL AT %M* : BOOL; //Driftfel fläkt~wp:	


	PV8 AT %M* : STRING;//Modbus konfiguering~wp:
	FAULT AT %M* : BOOL;//Kommunikationsfel~wp:
	
END_VAR
VAR
	
	offset : WORD;
	rTemp : REAL;
	iTemp : UINT;
	bSekvensFlagga : BOOL;
			
	FB_MBReadRegs_ArrHolding1: FB_MBReadRegs;
	ArrHolding1 : ARRAY [0..20] OF WORD; //Holding
		
	//Kommunikationsfel
	fbKommTof : tof; 
	fbKommTon : ton;
	
	sIP: STRING(255);
	sPort: STRING(255);
	sModbusID: STRING(255);
	sModbusLoop: STRING(255);
	sTemp : STRING(255);
	
	fbReadWriteHoldingReg01 : fbReadWriteHoldingReg;
	
	iWrite : INT;
END_VAR

//General
	offset := 0;
//Sekvens	
	bSekvensFlagga := oaksGVL.aBModbusSekvens[iModbusLoop] = UINT_TO_INT(nUnitID);
//Modbus konfiguering
	sIP := CONCAT (SIPAddr, '');
	sPort := CONCAT ('<br>Port: ', UINT_TO_STRING(nTCPPort)); 								
	sModbusID := CONCAT('<br>ID: ', UINT_TO_STRING(nUnitID));
	sModbusLoop := CONCAT('<br>Loop: ', INT_TO_STRING(iModbusLoop));	

	sTemp := sIP;
	sTemp := CONCAT(sTemp, sPort);
	sTemp := CONCAT(sTemp, sModbusID);
	sTemp := CONCAT(sTemp, sModbusLoop);
	
	PV8 := sTemp;

///////////////
//READ
///////////////

	iWrite := REAL_TO_INT(rSetpoint);
fbReadWriteHoldingReg01(
	sIPAddr:= sIpAddr, 
	nTCPPort:= INT_TO_UINT(nTCPPort), 
	nUnitID:= INT_TO_BYTE(nUnitID), 
	mBusAdr:=9 , 
	bEnable:= bSekvensFlagga, 
	iWrite:= INT_TO_UINT(iWrite), 
	iRead=> , 
	bError=> , 
	bBusy=> );
	
	//Read Holding 0-10
	FB_MBReadRegs_ArrHolding1(
	sIPAddr:= sIpAddr, 
	nTCPPort:= INT_TO_UINT(nTCPPort), 
	nUnitID:= INT_TO_BYTE(nUnitID), 
	nQuantity:= 12, 
	nMBAddr:= 0 + offset, 
	cbLength:= SIZEOF(ArrHolding1), 
	pDestAddr:= ADR(ArrHolding1), 
	bExecute:= bSekvensFlagga, 
	tTimeout:= T#3S, 
	bBusy=> , 
	bError=> , 
	nErrId=> , 
	cbRead=> );
	
		//Values
		//ArrHolding1[0]; //0
		PV := WORD_TO_REAL(ArrHolding1[1]); //1
		//ArrHolding1[2]; //2
		OP := WORD_TO_REAL(ArrHolding1[3]); //3
		rTemp :=  WORD_TO_REAL(ArrHolding1[4]);
		PV1 := rTemp / 10;
		//ArrHolding1[5]; //5
		//ArrHolding1[6]; //6
		AL := ArrHolding1[7] < 1; //7
		CSP := WORD_TO_REAL(ArrHolding1[8]); //8
		//ArrHolding1[8]; //9
		//ArrHolding1[8]; //10
		
	
//Communication error
	fbKommTof(IN:=FB_MBReadRegs_ArrHolding1.bError , PT:=T#20S , Q=> , ET=> );
	fbKommTon(IN:=fbKommTof.Q , PT:=T#20M , Q=> , ET=> );
	FAULT :=fbKommTon.Q;
		
//Write busy	
	oaksgvl.aBModbusBusyFlagga[iModbusLoop,nUnitID] := FB_MBReadRegs_Arrholding1.bBusy OR fbReadWriteHoldingReg01.bBusy;

END_FUNCTION_BLOCK

// oaksModbusLibrary/Datahantering/fbReadWriteHoldingReg
//OAKS AB
//2020-05-12
//Funktionsblock för läsning av holding register. Värde skrivs endast då skriv värde avviker från återläst värde. Används ej på EEPROM minnen, då det riskerar att skriva sönder dem. Använd istället block med återläsning av värden. 
{attribute 'obsolete' := 'Använd ersättningsblock fbReadWriteHoldingReal'}
FUNCTION_BLOCK fbReadWriteHoldingReg
VAR_INPUT
	sIPAddr : STRING := ''; 
	nTCPPort : UINT;
	nUnitID : UINT;
	mBusAdr : UINT;
	bEnable : BOOL := TRUE;
	iWrite : UINT; //Värde att skriva
	tTimeout : TIME := T#5S;
END_VAR

VAR_OUTPUT
	iRead : UINT; //Återläst värde
	bError : BOOL; //Felindikering från block
	bBusy : BOOL; //Funtionsblock upptaget
END_VAR

VAR
	fbReadRegs_1: FB_MBReadRegs;
	fbWriteSingleReg_1: FB_MBWriteSingleReg;

	nIdx: INT;
	R_TRIGstart : R_TRIG;
END_VAR

//Read Regs
					
		fbReadRegs_1(
			sIPAddr:= sIPAddr, 
			nTCPPort:= INT_TO_UINT(nTCPPort), 
			nUnitID:= INT_TO_BYTE(nUnitID), 
			nQuantity:= 1, 
			nMBAddr:= UINT_TO_WORD(mBusAdr), 
			cbLength:= SIZEOF(iRead), 
			pDestAddr:= ADR(iRead), 
			bExecute:= bEnable, 
			tTimeout:= tTimeout, 
			bBusy=> , 
			bError=> , 
			nErrId=> , 
			cbRead=> );

//Write regs
		
		IF iWrite <> iRead  AND NOT fbReadRegs_1.bBusy AND bEnable THEN
			fbWriteSingleReg_1.bExecute := TRUE;
		ELSE
			fbWriteSingleReg_1.bExecute := FALSE;
		END_IF
			
		fbWriteSingleReg_1(
			sIPAddr:= sIPAddr, 
			nTCPPort:= INT_TO_UINT(nTCPPort), 
			nUnitID:= INT_TO_BYTE(nUnitID), 
			nMBAddr:= UINT_TO_WORD(mBusAdr),
			nValue:= iWrite, 
			bExecute:= , //From if/else 
			tTimeout:= tTimeout , 
			bBusy=> , 
			bError=> , 
			nErrId=> );
			
		//Uptagen
		bBusy := fbReadRegs_1.bBusy OR fbWriteSingleReg_1.bBusy;
	
		//Fel
		bError := fbReadRegs_1.bError OR fbWriteSingleReg_1.bError;

END_FUNCTION_BLOCK

// oaksModbusLibrary/Calectro/fbCalectroIoMb02
//OAKS AB
//2020-05-12
//Påbörjat block för calectros io-låda. EJ KLART!!
FUNCTION_BLOCK fbCalectroIoMb02
VAR_INPUT
	sIPAddr : STRING := ''; 
	nTCPPort : UINT;
	nUnitID : UINT :=1;
	iModbusLoop : INT :=1; //Modbusslinga
	tTimeout : TIME := T#10S;
	DO1_CMD AT %M*	: BOOL;//Digital utgång 1~wp:[trendoptions]i:14400, t:1
	DO2_CMD AT %M*	: BOOL;//Digital utgång 2~wp:[trendoptions]i:14400, t:1
	AO1_OP AT %M*	: REAL;//Analog utgång 1~wp:[trendoptions]i:300
	AO2_OP AT %M*	: REAL;//Analog utgång 2~wp:[trendoptions]i:300
END_VAR
VAR_OUTPUT
	DI1_V AT %M*	: BOOL;//Digital ingång 1~wp:[trendoptions]i:14400, t:1
	DI2_V AT %M*	: BOOL;//Digital ingång 2~wp:[trendoptions]i:14400, t:1
	DI3_V AT %M*	: BOOL;//Digital ingång 3~wp:[trendoptions]i:14400, t:1
	DI4_V AT %M*	: BOOL;//Digital ingång 4~wp:[trendoptions]i:14400, t:1

	AI1_PV AT %M*	: REAL;//Analog ingång 1~wp:[trendoptions]i:300
	AI2_PV AT %M*	: REAL;//Analog ingång 2~wp:[trendoptions]i:300
	AI3_PV AT %M*	: REAL;//Analog ingång 3~wp:[trendoptions]i:300
	AI4_PV AT %M*	: REAL;//Analog ingång 4~wp:[trendoptions]i:300
	
	PV8 AT %M* : STRING;//Modbus konfiguering~wp:
	FAULT AT %M* : BOOL;//Kommunikationsfel~wp:
	
END_VAR
VAR
	offset : WORD;
	rTemp : REAL;
	iTemp : UINT;
	bSekvensFlagga : BOOL;
			
	FB_MBReadInputRegs_ArrHolding1: FB_MBReadInputRegs;
	ArrHolding1 : ARRAY [0..10] OF WORD; //Holding
		
	//Kommunikationsfel
	fbKommTof : tof; 
	fbKommTon : fbAlarm;
	
	sIP: STRING(255);
	sPort: STRING(255);
	sModbusID: STRING(255);
	sModbusLoop: STRING(255);
	sTemp : STRING(255);
	
	
	fbReadWriteHoldingRegAo1: fbReadWriteHoldingReg;
	fbReadWriteHoldingRegAo2: fbReadWriteHoldingReg;
END_VAR

//General
	offset := 0;
//Sekvens	
	bSekvensFlagga := oaksGVL.aBModbusSekvens[iModbusLoop] = UINT_TO_INT(nUnitID);
//Modbus konfiguering
	sIP := CONCAT (SIPAddr, '');
	sPort := CONCAT ('<br>Port: ', UINT_TO_STRING(nTCPPort)); 								
	sModbusID := CONCAT('<br>ID: ', UINT_TO_STRING(nUnitID));
	sModbusLoop := CONCAT('<br>Loop: ', INT_TO_STRING(iModbusLoop));	

	sTemp := sIP;
	sTemp := CONCAT(sTemp, sPort);
	sTemp := CONCAT(sTemp, sModbusID);
	sTemp := CONCAT(sTemp, sModbusLoop);
	
	PV8 := sTemp;

///////////////		
//READ
///////////////		
//4x0007 Analog output #1 x100 (Volt) /PWM x10 (%)0 to 1000
	fbReadWriteHoldingRegAo1(
	sIPAddr:= sIpAddr, 
	nTCPPort:= INT_TO_UINT(nTCPPort), 
	nUnitID:= INT_TO_BYTE(nUnitID), 
	mBusAdr:=6 , 
	tTimeout := tTimeout, 
	bEnable:=bSekvensFlagga , 
	iWrite:=REAL_TO_UINT(AO1_OP)*10 , 
	iRead=> , 
	bError=> , 
	bBusy=> );


//4x0008 Analog output #2 x100 (Volt) /PWM x10 (%)0 to 1000
	fbReadWriteHoldingRegAo2(
	sIPAddr:= sIpAddr, 
	nTCPPort:= INT_TO_UINT(nTCPPort), 
	nUnitID:= INT_TO_BYTE(nUnitID), 
	mBusAdr:=7 , 
	tTimeout := tTimeout, 
	bEnable:=bSekvensFlagga , 
	iWrite:=REAL_TO_UINT(AO1_OP)*10 , 
	iRead=> , 
	bError=> , 
	bBusy=> );


	
	//Read Holding 0-10
	FB_MBReadInputRegs_ArrHolding1(
	sIPAddr:= sIpAddr, 
	nTCPPort:= INT_TO_UINT(nTCPPort), 
	nUnitID:= INT_TO_BYTE(nUnitID), 
	nQuantity:= 4, 
	nMBAddr:= 16 + offset, 
	cbLength:= SIZEOF(ArrHolding1), 
	pDestAddr:= ADR(ArrHolding1), 
	bExecute:= bSekvensFlagga, 
	tTimeout:= tTimeout, 
	bBusy=> , 
	bError=> , 
	nErrId=> , 
	cbRead=> );
	
		//Values
		rTemp := ArrHolding1[0]; //0
		AI1_PV := rTemp / 10; //1
		rTemp := ArrHolding1[1]; //0
		AI2_PV := rTemp / 10; //1
		rTemp := ArrHolding1[2]; //0
		AI3_PV := rTemp / 10; //1
		rTemp := ArrHolding1[3]; //0
		AI4_PV := rTemp / 10; //1
		//ArrHolding1[4]; //4
		//ArrHolding1[5]; //5
		//ArrHolding1[6]; //6
		//ArrHolding1[7]; //7
		//ArrHolding1[8]; //8
		//ArrHolding1[9]; //9
		//ArrHolding1[10]; //10
		
	
//Communication error
	fbKommTof(IN:=FB_MBReadInputRegs_ArrHolding1.bError , PT:=T#20S , Q=> , ET=> );
	fbKommTon(bInput:=fbKommTof.Q , tAlarmDelay:=T#20M , bAutoReset:= , bAlarmOutput=> );
	FAULT :=fbKommTon.bAlarmOutput;
//Write busy	
	oaksgvl.aBModbusBusyFlagga[iModbusLoop,nUnitID] := FB_MBReadInputRegs_ArrHolding1.bBusy;

END_FUNCTION_BLOCK

// oaksModbusLibrary/Daikin/fbDaikinRTDNET
//Funktionsblock för kommunikation mot kom.modul Daikin RTD-NET (via ModbusTCP-gateway), för kommunikation med t ex luftvärmepumpar
//Robert H Oaks AB 
//22-03-14

//V 1.0		Endast läsning av värden, endast Group Feedback (unit feedback kan enkelt läggas till senare. Testad

//OBS! Ej anpassad för Modbus-sekvens i oaks-standard, bör åtgärdas!!

(*

I0021	Is Fault 0..1
I0022	Fault Code 0..65535
I0023	Return Air Average °C x100
I0024	Filter Alarm 0..1
I0030	Thermo On 0..3s
I0035	Defrost 0..1

*)



FUNCTION_BLOCK fbDaikinRTDNET
VAR_INPUT
	sIPAddr 		: STRING; 			//Ip-adress till ModbusTCP-gateway
	nMBTCPPort		: UINT := 502;		//ModbusTCP-port
	nUnitID			: UINT := 1;		//Enhetsadress
	tInterval		: TIME := T#10S;	//Kommunikationsintervall
	tTimeout		: TIME := T#3S;	//Timeout 
END_VAR

VAR_OUTPUT
	V		AT %M*		: BOOL;				//Driftindikering~wp:[trendoptions]i:14400, t:1
	PV		AT %M* 		: REAL; 			//Temperatur rumsluft~wp:[unit]°C[format]0.0[trendoptions]i:300
	PV1		AT %M* 		: STRING := ''; 	//Driftläge~wp:[trendoptions]i:14400, t:1
	FAULT	AT %M*		: BOOL;				//Summafel luftkonditionering~wp:[alarmoptions]p:3
	PV8		AT %M*		: UINT;				//Felkod (255 = Inget fel) ~wp:[trendoptions]i:14400, t:1
	AL1		AT %M*		: BOOL;				//Filterlarm luftkonditionering~wp:[alarmoptions]p:3
	V1		AT %M*		: BOOL;				//Avfrostning aktiv~wp:[trendoptions]i:14400, t:1
	AL8		AT %M*		: BOOL;				//Kommunikationsfel luftkonditionering~wp:[alarmoptions]p:3
END_VAR

VAR
	bRun			: BOOL;	
	fbRunTON		: TON;
	fbRunTRIG		: R_TRIG;

	fbReadI0021		: FB_MBReadInputRegs;
	fbReadI0022		: FB_MBReadInputRegs;
	fbReadI0023		: FB_MBReadInputRegs;
	fbReadI0024		: FB_MBReadInputRegs;
	fbReadI0030		: FB_MBReadInputRegs;
	fbReadI0035		: FB_MBReadInputRegs;

	wRead0021, wRead0022, wRead0023, wRead0024, wRead0030, wRead0035		: WORD;
	
	fbErrorTOF		: TOF;
	fbErrorTON		: TON;
END_VAR

fbRunTON(IN := NOT bRun, PT := tInterval);
fbRunTRIG(CLK := fbRunTON.Q, Q => bRun);

fbReadI0021(sIPAddr := sIPAddr, nTCPPort := nMBTCPPort, nUnitID := UINT_TO_BYTE(nUnitID), nQuantity := 1, bExecute := bRun, tTimeout := tTimeout,   
	nMBAddr 	:= 21,
	cbLength	:= SIZEOF(wRead0021),
	pDestAddr	:= ADR(wRead0021));
	FAULT := wRead0021 > 0;
	
fbReadI0022(sIPAddr := sIPAddr, nTCPPort := nMBTCPPort, nUnitID := UINT_TO_BYTE(nUnitID), nQuantity := 1, bExecute := bRun, tTimeout := tTimeout,   
	nMBAddr 	:= 22,
	cbLength	:= SIZEOF(wRead0022),
	pDestAddr	:= ADR(wRead0022));
	PV8 := wRead0022;
	
fbReadI0023(sIPAddr := sIPAddr, nTCPPort := nMBTCPPort, nUnitID := UINT_TO_BYTE(nUnitID), nQuantity := 1, bExecute := bRun, tTimeout := tTimeout,   
	nMBAddr 	:= 23,
	cbLength	:= SIZEOF(wRead0023),
	pDestAddr	:= ADR(wRead0023));
	PV := INT_TO_REAL(WORD_TO_INT(wRead0023)) / 100;
	
fbReadI0024(sIPAddr := sIPAddr, nTCPPort := nMBTCPPort, nUnitID := UINT_TO_BYTE(nUnitID), nQuantity := 1, bExecute := bRun, tTimeout := tTimeout,   
	nMBAddr 	:= 24,
	cbLength	:= SIZEOF(wRead0024),
	pDestAddr	:= ADR(wRead0024));
	AL1 := wRead0024 > 0;
	
fbReadI0030(sIPAddr := sIPAddr, nTCPPort := nMBTCPPort, nUnitID := UINT_TO_BYTE(nUnitID), nQuantity := 1, bExecute := bRun, tTimeout := tTimeout,   
	nMBAddr 	:= 30,
	cbLength	:= SIZEOF(wRead0030),
	pDestAddr	:= ADR(wRead0030));
	
	CASE wRead0030 OF 
		0:
		PV1	:= 'Standby';
		1:
		PV1	:= 'Värme';
		2:
		PV1	:= 'Kyla';
		3:
		PV1	:= 'Värme/kyla';
	END_CASE;
	
	V := wRead0030 > 0;
	
fbReadI0035(sIPAddr := sIPAddr, nTCPPort := nMBTCPPort, nUnitID := UINT_TO_BYTE(nUnitID), nQuantity := 1, bExecute := bRun, tTimeout := tTimeout,   
	nMBAddr 	:= 35,
	cbLength	:= SIZEOF(wRead0035),
	pDestAddr	:= ADR(wRead0035));
	V1 := wRead0035 > 0;
	

//Kom.fel modbus
fbErrorTOF(IN := fbReadI0021.bError, PT := T#30S);
fbErrorTON(IN := fbErrorTOF.Q, PT := T#120S, Q => AL8);

END_FUNCTION_BLOCK

// oaksModbusLibrary/Danfoss/fbDanfossDGS_HFC
//Funktionsblock för kommunikation mot Danfoss DGS-HFC gasgivare via basenhet (via ModbusTCP-gateway). 
//OBS, kritiskt gaslarm ej i detta block, ska köras hårdtrådat
//Robert H Oaks AB 
//22-03-21

//V 1.0	Testad

//OBS! Ej anpassad för Modbus-sekvens i oaks-standard, bör åtgärdas!!

(*

Common errors 10064
Crit. limit ppm 10080
Warn. limit ppm 10094
Alarm delay s 10061
Reset alarm 10065
Reset alarm time 10091
DGS Warm-up 10089
Days till calib 10090
Rem. sensivity 10092
Out of range 20002
Wrong SensorType 20003
Sensor removed 20004
Calibrate sensor 20005
Warning limit 20006
*)



FUNCTION_BLOCK fbDanfossDGS_HFC
VAR_INPUT
	sIPAddr 		: STRING; 			//Ip-adress till ModbusTCP-gateway
	nMBTCPPort		: UINT := 502;		//ModbusTCP-port
	nUnitID			: UINT := 1;		//Enhetsadress
	tInterval		: TIME := T#10S;	//Kommunikationsintervall
	tTimeout		: TIME := T#3S;		//Timeout
	AHHL AT %M*		: REAL;				//Larmgräns kritisk gasnivå ~wp:[unit]ppm[format]0[trendoptions]i:60
	AHL AT %M*		: REAL;				//Larmgräns hög gasnivå ~wp:[unit]ppm[format]0[trendoptions]i:60 
	AD AT %M*		: REAL;				//Larmfördröjning gasnivå ~wp:[unit]s[format]0[trendoptions]i:60
	CMD AT %M*		: BOOL;				//Reset/blockering gaslarm ~wp: 
	SP1 AT %M*		: REAL;				//Larmblockeringstid vid kvittering ~wp:[unit]s[format]0[trendoptions]i:60
END_VAR

VAR_OUTPUT
	V1		AT %M* 		: BOOL; 			//Uppvärmningsläge ~wp:[trendoptions]i:14400, t:1
	PV1		AT %M* 		: UINT; 			//Tid kvar nästa kalibrering ~wp:[unit]dagar[format]0[trendoptions]i:300
	PV2		AT %M* 		: UINT; 			//Återstående livslängd ~wp:[unit]%[format]0[trendoptions]i:300
	FAULT	AT %M*		: BOOL;				//Summalarm givarfel~wp:[alarmoptions]p:1
	AL1		AT %M*		: BOOL;				//Kalibrering av givare nödvändig~wp:[alarmoptions]p:3
	AL2		AT %M*		: BOOL;				//Summalarm basenhet~wp:[alarmoptions]p:2
	HL		AT %M*		: BOOL;				//Larm hög gasnivå (ej kritisk)~wp:[alarmoptions]p:2
	AL8		AT %M*		: BOOL;				//Kommunikationsfel basenhet gasgivare~wp:[alarmoptions]p:1
END_VAR

VAR
	bRun			: BOOL;	
	fbRunTON		: TON;
	fbRunTRIG		: R_TRIG;
	
	fbRW10061		: fbHoldingRWReadBackEEPROM_REAL;
	fbRW10065		: fbHoldingRWReadBackEEPROM_BOOL;
	fbRW10080		: fbHoldingRWReadBackEEPROM_REAL;
	fbRW10091		: fbHoldingRWReadBackEEPROM_REAL;
	fbRW10094		: fbHoldingRWReadBackEEPROM_REAL;
	
	fbRead10064		: FB_MBReadRegs;
	fbRead10089		: FB_MBReadRegs;
	fbRead10090		: FB_MBReadRegs;
	fbRead10092		: FB_MBReadRegs;
	fbRead20002_4	: FB_MBReadRegs;
	fbRead20005		: FB_MBReadRegs;
	fbRead20006		: FB_MBReadRegs;
	
	
	wRead10064, wRead10089, wRead10090, wRead10092, wRead20005, wRead20006		: WORD;
	awRead20002_4 : ARRAY[0..2] OF WORD;
	
	fbErrorTOF		: TOF;
	fbErrorTON		: TON;
	
END_VAR

fbRunTON(IN := NOT bRun, PT := tInterval);
fbRunTRIG(CLK := fbRunTON.Q, Q => bRun);

(* Läs/skriv värden *)

//Reset alarm 10065		Reset & blockering av larm
fbRW10065(sIPAddr := sIPAddr, nMBTCPPort := nMBTCPPort, nUnitID := nUnitID, tTimeout := tTimeout, bRun := bRun,
		nMBAddr := 10064,
	 	bValue	:= CMD);
		
//Reset alarm time 10091	Tid för larmblockering vid larmreset		
fbRW10091(sIPAddr := sIPAddr, nMBTCPPort := nMBTCPPort, nUnitID := nUnitID, tTimeout := tTimeout, bRun := bRun,
		nMBAddr := 10090,
	 	rValue	:= SP1,
		uiScale	:= 1);	

//Crit. limit ppm 10080	Larmgräns kritisk gasnivå		
fbRW10080(sIPAddr := sIPAddr, nMBTCPPort := nMBTCPPort, nUnitID := nUnitID, tTimeout := tTimeout, bRun := bRun,
		nMBAddr := 10079,
	 	rValue	:= AHHL,
		uiScale	:= 1);		
		
//Warn. limit ppm 10094	Larmgräns hög gasnivå		
fbRW10094(sIPAddr := sIPAddr, nMBTCPPort := nMBTCPPort, nUnitID := nUnitID, tTimeout := tTimeout, bRun := bRun,
		nMBAddr := 10093,
	 	rValue	:= AHL,
		uiScale	:= 1);		
		
//Alarm delay s 10061		Fördröjning gaslarm hög/kritisk		
fbRW10061(sIPAddr := sIPAddr, nMBTCPPort := nMBTCPPort, nUnitID := nUnitID, tTimeout := tTimeout, bRun := bRun,
		nMBAddr := 10060,
	 	rValue	:= AD,
		uiScale	:= 1);		
	
		
(* Läs värden *)

//Common errors 10064		Summalarm från basenhet	
fbRead10064(sIPAddr := sIPAddr, nTCPPort := nMBTCPPort, nUnitID := UINT_TO_BYTE(nUnitID), nQuantity := 1, bExecute := bRun, tTimeout := tTimeout,   
	nMBAddr 	:= 10063,
	cbLength	:= SIZEOF(wRead10064),
	pDestAddr	:= ADR(wRead10064));
	AL2 := wRead10064 > 0;
	
//DGS Warm-up 10089			Uppvärmning givare	
fbRead10089(sIPAddr := sIPAddr, nTCPPort := nMBTCPPort, nUnitID := UINT_TO_BYTE(nUnitID), nQuantity := 1, bExecute := bRun, tTimeout := tTimeout,   
	nMBAddr 	:= 10088,
	cbLength	:= SIZEOF(wRead10089),
	pDestAddr	:= ADR(wRead10089));
	V1 := wRead10089 > 0;

//Days till calib 10090		Dagar kvar till kalibrering	
fbRead10090(sIPAddr := sIPAddr, nTCPPort := nMBTCPPort, nUnitID := UINT_TO_BYTE(nUnitID), nQuantity := 1, bExecute := bRun, tTimeout := tTimeout,   
	nMBAddr 	:= 10089,
	cbLength	:= SIZEOF(wRead10090),
	pDestAddr	:= ADR(wRead10090));
	PV1 := wRead10090;
	
//Rem. sensivity 10092		Återstående livslängd	
fbRead10092(sIPAddr := sIPAddr, nTCPPort := nMBTCPPort, nUnitID := UINT_TO_BYTE(nUnitID), nQuantity := 1, bExecute := bRun, tTimeout := tTimeout,   
	nMBAddr 	:= 10091,
	cbLength	:= SIZEOF(wRead10092),
	pDestAddr	:= ADR(wRead10092));
	PV2 := MIN(100, wRead10092);

//Out of range 20002, Wrong SensorType 20003, Sensor removed 20004		Summalarm givarfel		
fbRead20002_4(sIPAddr := sIPAddr, nTCPPort := nMBTCPPort, nUnitID := UINT_TO_BYTE(nUnitID), bExecute := bRun, tTimeout := tTimeout,
	nQuantity 	:= 3,   
	nMBAddr 	:= 20001,
	cbLength	:= SIZEOF(awRead20002_4),
	pDestAddr	:= ADR(awRead20002_4));
	FAULT := (awRead20002_4[0] > 0) OR (awRead20002_4[1] > 0) OR (awRead20002_4[2] > 0);

//Calibrate sensor 20005	Kalibreringslarm givare
fbRead20005(sIPAddr := sIPAddr, nTCPPort := nMBTCPPort, nUnitID := UINT_TO_BYTE(nUnitID), nQuantity := 1, bExecute := bRun, tTimeout := tTimeout,   
	nMBAddr 	:= 20004,
	cbLength	:= SIZEOF(wRead20005),
	pDestAddr	:= ADR(wRead20005));
	AL1 := wRead20005 > 0;	
	
//Warning limit 20006		Larm hög gasnivå (ej kritisk)
fbRead20006(sIPAddr := sIPAddr, nTCPPort := nMBTCPPort, nUnitID := UINT_TO_BYTE(nUnitID), nQuantity := 1, bExecute := bRun, tTimeout := tTimeout,   
	nMBAddr 	:= 20005,
	cbLength	:= SIZEOF(wRead20006),
	pDestAddr	:= ADR(wRead20006));
	HL := wRead20006 > 0;	

//Kom.fel modbus
fbErrorTOF(IN := fbRead20006.bError, PT := T#30S);
fbErrorTON(IN := fbErrorTOF.Q, PT := T#120S, Q => AL8);

END_FUNCTION_BLOCK

// oaksModbusLibrary/Datahantering/fbHoldingRWReadBackEEPROM_REAL
// Funktionsblock för att läsa/skriva enskilda holdingregister, med återläsning och skrivspärr för att skydda EEPROM. Skrivspärr från överordnat block
// Datatyp REAL -> WORD med skalning
FUNCTION_BLOCK fbHoldingRWReadBackEEPROM_REAL
VAR_INPUT
	sIPAddr 		: STRING; 			
	nMBTCPPort		: UINT;		
	nUnitID			: UINT;
	nMBAddr			: UINT;
	tTimeout		: TIME;
	bRun			: BOOL;
	bWriteBlock		: BOOL;
	uiScale			: UINT := 1;
END_VAR

VAR_IN_OUT
	rValue			: REAL;
END_VAR
VAR_OUTPUT
	bComError		: BOOL;
	bSyncError		: BOOL;
	bWBusy			: BOOL;
END_VAR
VAR
	fbRead			: FB_MBReadRegs;
	fbWrite			: FB_MBWriteSingleReg;
	
	fbSyncErrorTON	: TON;
	
	wReadMaster		: WORD;
	wOldReadMaster	: WORD;
	wReadSlave		: WORD;
	wOldReadSlave	: WORD;
	
	bMasterValChgd	: BOOL;
	bSlaveValChgd	: BOOL;
	bDidWrite		: BOOL;
	
	bInit			: BOOL := TRUE;
	fbInitTON		: TON;
	iCase			: INT;
	
	iKoll : INT;
END_VAR

// Vid uppstart vänta 5s, läs endast slavvärdet
IF bInit THEN
	fbInitTON(IN := TRUE, PT := T#5S);
	
	fbRead(sIPAddr := sIPAddr, nTCPPort := nMBTCPPort, nUnitID := UINT_TO_BYTE(nUnitID), nQuantity := 1, bExecute := bRun, tTimeout := tTimeout,   
				nMBAddr 	:= nMBAddr,
				cbLength	:= SIZEOF(wReadSlave),
				pDestAddr	:= ADR(wReadSlave));
	
	IF fbInitTON.Q THEN
		bInit := FALSE;
	END_IF
	
ELSE

	IF uiScale = 0 THEN
		uiScale := 1;
	END_IF
	
	// Läs lokalt värde och kontrollera ev ändring av värde
	wReadMaster 	:= REAL_TO_UINT(rValue * uiScale);
	bMasterValChgd	:= wReadMaster <> wOldReadMaster;
	
	
	// Läs värde från modbus-slav och kontrollera ev ändring av värde
	fbRead(sIPAddr := sIPAddr, nTCPPort := nMBTCPPort, nUnitID := UINT_TO_BYTE(nUnitID), nQuantity := 1, bExecute := bRun, tTimeout := tTimeout,   
				nMBAddr 	:= nMBAddr,
				cbLength	:= SIZEOF(wReadSlave),
				pDestAddr	:= ADR(wReadSlave));
				
	bSlaveValChgd	:= wReadSlave <> wOldReadSlave;
	
	// Om slav-värde ändrats, uppdatera in-ut-värde och kontrollvärden så att ingen återskrivning sker
	IF bSlaveValChgd THEN
		rValue 			:= UINT_TO_REAL(wReadSlave) / uiScale;
		wReadMaster 	:= wReadSlave;
		wOldReadMaster 	:= wReadSlave;
		wOldReadSlave	:= wReadSlave;
	END_IF
	
	bDidWrite := FALSE;	// Initiera flagga
	// Om master-värde ändrats:
	IF bMasterValChgd AND NOT fbRead.bError AND NOT bWriteBlock THEN
		CASE iCase OF
			0:
				
			fbWrite(sIPAddr := sIPAddr, nTCPPort := nMBTCPPort, nUnitID := UINT_TO_BYTE(nUnitID), tTimeout := tTimeout,		// Skriv värdet
						bExecute 	:= bRun,   
						nMBAddr 	:= nMBAddr,
						nValue		:= wReadMaster);
			
			IF fbWrite.bBusy THEN						
				bDidWrite := TRUE;	// Sätt flagga för utförd skrivning
			END_IF;
			
			IF NOT fbWrite.bBusy AND NOT fbWrite.bError AND bDidWrite THEN
				iCase := 1;
			END_IF
			
			1:
			
			IF wReadSlave = wReadMaster THEN	// Vänta på att värde från slav stämmer med skrivet värde
				iKoll	:= iKoll +1;
				bMasterValChgd 		:= FALSE;	// Återställ flagga för ändrat master-värde, uppdatera old-värde, återställ flaggor etc
				wOldReadMaster 		:= wReadMaster;
				bDidWrite 			:= FALSE;
				iCase := 0;
			END_IF
		
		END_CASE
	END_IF
	
	fbWrite();
	
	fbSyncErrorTON(IN := bDidWrite, PT := T#60S, Q => bSyncError);	// Om skrivning skett och inte återläst värde är samma inom 60sek, sätt flagga för synkfel
	
	bWBusy := fbWrite.bBusy;	// Visa att skrivblocket är aktivt, för att överordnad funktion ska kunna hantera begränsning av skrivning
	bComError := fbRead.bError;
	
END_IF;

END_FUNCTION_BLOCK

// oaksModbusLibrary/Datahantering/fbHoldingRWReadBackEEPROM_BOOL
//Funktionsblock för att läsa/skriva enskilda holdingregister, med återläsning och skrivspärr för att skydda EEPROM. Skrivspärr från överordnat block
//Datatyp BOOL -> WORD (en BOOL per helt dataord)
FUNCTION_BLOCK fbHoldingRWReadBackEEPROM_BOOL
VAR_INPUT
	sIPAddr 		: STRING; 			
	nMBTCPPort		: UINT;		
	nUnitID			: UINT;
	nMBAddr			: UINT;
	tTimeout		: TIME;
	bRun			: BOOL;
	bWriteBlock		: BOOL;
END_VAR

VAR_IN_OUT
	bValue			: BOOL;
END_VAR
VAR_OUTPUT
	bComError		: BOOL;
	bSyncError		: BOOL;
	bWBusy			: BOOL;
END_VAR
VAR
	fbRead			: FB_MBReadRegs;
	fbWrite			: FB_MBWriteSingleReg;
	
	fbSyncErrorTON	: TON;
	
	wReadMaster		: WORD;
	wOldReadMaster	: WORD;
	wReadSlave		: WORD;
	wOldReadSlave	: WORD;
	
	bMasterValChgd	: BOOL;
	bSlaveValChgd	: BOOL;
	bDidWrite		: BOOL;
END_VAR

//Läs lokalt värde och kontrollera ev ändring av värde
wReadMaster 	:= BOOL_TO_WORD(bValue);
bMasterValChgd	:= wReadMaster <> wOldReadMaster;


//Läs värde från modbus-slav och kontrollera ev ändring av värde
fbRead(sIPAddr := sIPAddr, nTCPPort := nMBTCPPort, nUnitID := UINT_TO_BYTE(nUnitID), nQuantity := 1, bExecute := bRun, tTimeout := tTimeout,   
			nMBAddr 	:= nMBAddr,
			cbLength	:= SIZEOF(wReadSlave),
			pDestAddr	:= ADR(wReadSlave));
			
bSlaveValChgd	:= wReadSlave <> wOldReadSlave;

//Om slav-värde ändrats, uppdatera in-ut-värde och kontrollvärden så att ingen återskrivning sker
IF bSlaveValChgd THEN
	bValue 			:= WORD_TO_BOOL(wReadSlave);
	wReadMaster 	:= wReadSlave;
	wOldReadMaster 	:= wReadSlave;
	wOldReadSlave	:= wReadSlave;
END_IF

//Om master-värde ändrats:
IF bMasterValChgd THEN
	IF NOT fbWrite.bBusy AND NOT fbRead.bError AND NOT bDidWrite AND NOT bWriteBlock THEN		//Om skrivning redan aktiv, om ej redan skrivit och om skrivning ej blockerad:
		fbWrite(sIPAddr := sIPAddr, nTCPPort := nMBTCPPort, nUnitID := UINT_TO_BYTE(nUnitID), tTimeout := tTimeout,		//Skriv värdet
					bExecute 	:= TRUE,   
					nMBAddr 	:= nMBAddr,
					nValue		:= wReadMaster);
					
		bDidWrite := TRUE;	//Sätt flagga för utförd skrivning
	ELSE	
		IF wReadSlave = wReadMaster THEN	//Vänta på att värde från slav stämmer med skrivet värde
			bMasterValChgd 		:= FALSE;	//Återställ flagga för ändrat master-värde, uppdatera old-värde, återställ flaggor etc
			wOldReadMaster 		:= wReadMaster;
			bDidWrite 			:= FALSE;
			fbWrite.bExecute	:= FALSE;
		ELSE								//Om inte värde synkats, utför ny skrivning enligt intervalltimer
			IF bRun AND NOT fbWrite.bBusy THEN
				bDidWrite 			:= FALSE;
				fbWrite.bExecute	:= FALSE;
			END_IF
		END_IF
	END_IF
	
END_IF

fbSyncErrorTON(IN := bMasterValChgd, PT := T#10S, Q => bSyncError);	//Om skrivning skett och inte återläst värde är samma inom 10sek, sätt flagga för synkfel

fbWrite();	//Kör block för att uppdatera status

bWBusy := fbWrite.bBusy;	//Visa att skrivblocket är aktivt, för att överordnad funktion ska kunna hantera begränsning av skrivning
bComError := fbRead.bError;

END_FUNCTION_BLOCK

// oaksModbusLibrary/Danfoss/fbDanfossEKE347
//Funktionsblock för kommunikation mot Danfoss nivåcontroller EKE347 (via ModbusTCP-gateway) för t ex reglering av expansionsventiler i kylmaskiner.
//Med funktion för att skydda EEPROM mot sönderskrivning (max 10 skrivningar per minut tillåtet)
//Robert H Oaks AB 
//22-03-17

//V 1.0	Testad

//OBS! Ej anpassad för Modbus-sekvens i oaks-standard, bör åtgärdas!!

(*

r12 Main switch				3001
R01 Liquid level setpoint	3002
a02 Lower level limit		3004
a01 Upper level limit		3005
a04 Lower delay				3007
a03 Upper delay				3008
a12 Oscillation detect band	3012
a13 Oscillation detect tmut	3013	
n04 P-band					3016
n05 Integration time Tn		3017
n34 Neutral zone			3018
n32 Maximum OD				3022

B01 Controller state		4001
u01 Actual level			4002
u02 Actual reference		4003
u24 Actual OD				4004
u33 Actual valve position	4005

A1 Upper level				1901.8
A2 Lower level				1901.9
A92 Oscillation in level si	1901.10
A96 Valve position			1901.14
E1 Internal error			1901.0
E96 AKS 4100 error			1901.3
*)



FUNCTION_BLOCK fbDanfossEKE347
VAR_INPUT
	sIPAddr 		: STRING; 			//Ip-adress till ModbusTCP-gateway
	nMBTCPPort		: UINT := 502;		//ModbusTCP-port
	nUnitID			: UINT := 1;		//Enhetsadress
	tInterval		: TIME := T#6S;		//Kommunikationsintervall
	tTimeout		: TIME := T#5S;		//Timeout
END_VAR;
VAR_IN_OUT	
	bMainSw 			: BOOL;				//Start nivåregulator
	rReferece			: REAL;				//Börvärde vätskenivå
	rLowLimit			: REAL;				//Gräns låg vätskenivå
	rHighLimit			: REAL;				//Gräns hög vätskenivå
	rADLowLimit			: REAL;				//Larmfördröjning låg nivå
	rADHighLimit		: REAL;				//Larmfördröjning hög nivå
	rOscBand			: REAL;				//Reglerområde oscillationsövervakning
	rOscTimeout			: REAL;				//Tidsgräns oscillationsövervakning
	rPband				: REAL;				//P-band regulator
	rItime				: REAL;				//I-tid regulator
	rNeutralZone		: REAL;				//Neutralzon regulator
	rMinOD				: REAL;				//Min tillåten öppningsgrad ventil
	rMaxOD				: REAL;				//Max tillåten öppningsgrad ventil	 
END_VAR

VAR_OUTPUT
	PV1 AT %M*		: STRING :='';		//Driftläge ~wp:[trendoptions]i:60
	nState			: UINT;				//Driftläge numeriskt (för program)
	rActLevel		: REAL;				//Aktuell vätskenivå
	rActReference	: REAL;				//Aktuellt börvärde
	rActOD			: REAL;				//Aktuell öppningsgrad ventil
	rActVP			: REAL;				//Aktuell ventilposition
	bAlarmHL			: BOOL;				//Larm hög vätskenivå
	bAlarmLL			: BOOL;				//Larm låg vätskenivå
	bAlarmOsc		: BOOL;				//Larm ojämn vätskenivå
	bAlarmVP			: BOOL;				//Larm felaktigt ventilläge
	
	FAULT AT %M*	: BOOL;				//Larm systemfel reglercentral ~wp:[alarmoptions]p:2
	
	//AL3 AT %M*		: BOOL;				//Larm nivågivarfel ~wp:[alarmoptions]p:1
	bSensorFault	: BOOL;				//Larm nivågivarfel
	AL8 AT %M*		: BOOL;				//Kommunikationsfel modbus ~wp:[alarmoptions]p:1
	AL4 AT %M*		: BOOL;				//Synkroniseringsfel vid skrivning modbus ~wp:[alarmoptions]p:1
	V1	 AT %M*		: BOOL;				//Skrivning blockerad för att skydda EEPROM ~wp:[trendoptions]i:14400, t:1
END_VAR

VAR
	bRun			: BOOL;	
	fbRunTON		: TON;
	fbRunTRIG		: R_TRIG;
	bWBusy			: BOOL;
	fbWriteRT		: R_TRIG;
	iWriteCNT		: INT;
	fbWriteMonTOF	: TOF;
	
	fbRW3001		: fbHoldingRWReadBackEEPROM_BOOL;
	fbRW3002		: fbHoldingRWReadBackEEPROM_REAL;
	fbRW3004		: fbHoldingRWReadBackEEPROM_REAL;
	fbRW3005		: fbHoldingRWReadBackEEPROM_REAL;
	fbRW3007		: fbHoldingRWReadBackEEPROM_REAL;
	fbRW3008		: fbHoldingRWReadBackEEPROM_REAL;
	fbRW3012		: fbHoldingRWReadBackEEPROM_REAL;
	fbRW3013		: fbHoldingRWReadBackEEPROM_REAL;
	fbRW3016		: fbHoldingRWReadBackEEPROM_REAL;
	fbRW3017		: fbHoldingRWReadBackEEPROM_REAL;
	fbRW3018		: fbHoldingRWReadBackEEPROM_REAL;
	fbRW3021		: fbHoldingRWReadBackEEPROM_REAL;
	fbRW3022		: fbHoldingRWReadBackEEPROM_REAL;
	
	fbR4001			: FB_MBReadRegs;
	fbR4002			: FB_MBReadRegs;
	fbR4003			: FB_MBReadRegs;
	fbR4004			: FB_MBReadRegs;
	fbR4005			: FB_MBReadRegs;
	fbR1901			: FB_MBReadRegs;
	
	wR4001			: WORD;
	wR4002			: WORD;
	wR4003			: WORD;
	wR4004			: WORD;
	wR4005			: WORD;
	wR1901			: WORD;
	
	fbErrorTOF		: TOF;
	fbErrorTON		: TON;
	
END_VAR

(* Läsintervallsfunktion *)
fbRunTON(IN := NOT bRun, PT := tInterval);
fbRunTRIG(CLK := fbRunTON.Q, Q => bRun);


(* Skrivövervakning; sätter blockeringsflagga till skrivblock om fler än 10 skrivningar skett inom en minut. Flaggan återställs när timern gått ut. *)
//Övervaka busy-flagga från samtliga skrivblock
bWBusy 	:= fbRW3001.bWBusy OR fbRW3002.bWBusy OR fbRW3004.bWBusy OR fbRW3005.bWBusy OR fbRW3007.bWBusy OR fbRW3008.bWBusy OR fbRW3012.bWBusy OR fbRW3013.bWBusy
		OR fbRW3016.bWBusy OR fbRW3017.bWBusy OR fbRW3018.bWBusy OR fbRW3022.bWBusy;

fbWriteMonTOF(IN := bWBusy AND NOT fbWriteMonTOF.Q, PT := T#1M);	//Om något block är busy, starta intervalltimer och övervaka stigande flank
fbWriteRT(CLK := bWBusy);

IF fbWriteMonTOF.Q THEN				//Om intervalltimern är aktiv, räkna antal gånger skrivblock blir aktiva
	IF fbWriteRT.Q THEN
		iWriteCNT := iWriteCNT + 1;
	END_IF;
	
	IF iWriteCNT >= 10 THEN			//Om 10 skrivningar eller mer under intervalltiden, sätt skrivblockering
		V1 := TRUE;
		iWriteCNT := 0;
	END_IF
ELSE
	iWriteCNT := 0;
	V1 := FALSE;
END_IF


(* Läs/skriv inställningar *)

//r12 Main switch 3001				Regulator från/till
fbRW3001(sIPAddr := sIPAddr, nMBTCPPort := nMBTCPPort, nUnitID := nUnitID, tTimeout := tTimeout, bRun := bRun, bWriteBlock := V1,
		nMBAddr := 3000,
	 	bValue	:= bMainSw);

//R01 Liquid level setpoint //	Börvärde vätskenivå		
fbRW3002(sIPAddr := sIPAddr, nMBTCPPort := nMBTCPPort, nUnitID := nUnitID, tTimeout := tTimeout, bRun := bRun, bWriteBlock := V1, 
		nMBAddr := 3001,
	 	rValue	:= rReferece,
		uiScale	:= 10);		
		
//a02 Lower level limit 3004		Låg gräns vätskenivå		
fbRW3004(sIPAddr := sIPAddr, nMBTCPPort := nMBTCPPort, nUnitID := nUnitID, tTimeout := tTimeout, bRun := bRun, bWriteBlock := V1, 
		nMBAddr := 3003,
	 	rValue	:= rLowLimit,
		uiScale	:= 1);
		
//a03 Upper level limit 3005		Hög gräns vätskenivå		
fbRW3005(sIPAddr := sIPAddr, nMBTCPPort := nMBTCPPort, nUnitID := nUnitID, tTimeout := tTimeout, bRun := bRun, bWriteBlock := V1, 
		nMBAddr := 3004,
	 	rValue	:= rHighLimit,
		uiScale	:= 1);

//a04 Lower delay 3007				Larmfördröjning låg nivå		
fbRW3007(sIPAddr := sIPAddr, nMBTCPPort := nMBTCPPort, nUnitID := nUnitID, tTimeout := tTimeout, bRun := bRun, bWriteBlock := V1, 
		nMBAddr := 3006,
	 	rValue	:= rADLowLimit,
		uiScale	:= 1);

//a05 Upper delay 3008				Larmfördröjning låg nivå		
fbRW3008(sIPAddr := sIPAddr, nMBTCPPort := nMBTCPPort, nUnitID := nUnitID, tTimeout := tTimeout, bRun := bRun, bWriteBlock := V1, 
		nMBAddr := 3007,
	 	rValue	:= rADHighLimit,
		uiScale	:= 1);

//a12 Oscillation detect band 3012	Reglerområde oscillationsövervakning		
fbRW3012(sIPAddr := sIPAddr, nMBTCPPort := nMBTCPPort, nUnitID := nUnitID, tTimeout := tTimeout, bRun := bRun, bWriteBlock := V1, 
		nMBAddr := 3011,
	 	rValue	:= rOscBand,
		uiScale	:= 1);
		
//a13 Oscillation detect tmut 3013	Tidsgräns oscillationsövervakning	
fbRW3013(sIPAddr := sIPAddr, nMBTCPPort := nMBTCPPort, nUnitID := nUnitID, tTimeout := tTimeout, bRun := bRun, bWriteBlock := V1, 
		nMBAddr := 3012,
	 	rValue	:= rOscTimeout,
		uiScale	:= 1);

//n04 P-band 3016					P-pand 
fbRW3016(sIPAddr := sIPAddr, nMBTCPPort := nMBTCPPort, nUnitID := nUnitID, tTimeout := tTimeout, bRun := bRun, bWriteBlock := V1, 
		nMBAddr := 3015,
	 	rValue	:= rPband,
		uiScale	:= 10);
		
//n05 Integration time Tn 3017		I-tid regulator
fbRW3017(sIPAddr := sIPAddr, nMBTCPPort := nMBTCPPort, nUnitID := nUnitID, tTimeout := tTimeout, bRun := bRun, bWriteBlock := V1, 
		nMBAddr := 3016,
	 	rValue	:= rItime,
		uiScale	:= 1);
		
//n34 Neutral zone 3018				Neutralzon regulator
fbRW3018(sIPAddr := sIPAddr, nMBTCPPort := nMBTCPPort, nUnitID := nUnitID, tTimeout := tTimeout, bRun := bRun, bWriteBlock := V1, 
		nMBAddr := 3017,
	 	rValue	:= rNeutralZone,
		uiScale	:= 10);

//n33 Minimum OD 3021				Min öppningsgrad ventil
fbRW3021(sIPAddr := sIPAddr, nMBTCPPort := nMBTCPPort, nUnitID := nUnitID, tTimeout := tTimeout, bRun := bRun, bWriteBlock := V1, 
		nMBAddr := 3020,
	 	rValue	:= rMinOD,
		uiScale	:= 1);
		
//n32 Maximum OD 3022				Max öppningsgrad ventil
fbRW3022(sIPAddr := sIPAddr, nMBTCPPort := nMBTCPPort, nUnitID := nUnitID, tTimeout := tTimeout, bRun := bRun, bWriteBlock := V1, 
		nMBAddr := 3021,
	 	rValue	:= rMaxOD,
		uiScale	:= 1);

//Larm återskrivningsfel
AL4 := 	fbRW3001.bSyncError OR fbRW3002.bSyncError OR fbRW3004.bSyncError OR fbRW3005.bSyncError OR fbRW3007.bSyncError OR fbRW3008.bSyncError OR
		fbRW3012.bSyncError OR fbRW3013.bSyncError OR fbRW3016.bSyncError OR fbRW3017.bSyncError OR fbRW3018.bSyncError OR fbRW3022.bSyncError;

(* Läs värden *)
//B01 Controller state 4001			Driftläge regulator	
fbR4001(sIPAddr := sIPAddr, nTCPPort := nMBTCPPort, nUnitID := UINT_TO_BYTE(nUnitID), nQuantity := 1, bExecute := bRun, tTimeout := tTimeout,   
	nMBAddr 	:= 4000,
	cbLength	:= SIZEOF(wR4001),
	pDestAddr	:= ADR(wR4001));
	nState		:= wR4001;
	
IF fbR4001.bError THEN
	PV1 := 'Offline';
ELSE	
	CASE wR4001 OF 
		0:
		PV1	:= 'Uppstart';
		1:
		PV1	:= 'Stand-by';
		2:
		PV1	:= 'Auto/normal';
		3:
		PV1	:= 'Manuell';
		4:
		PV1	:= 'Slav';
		5:
		PV1	:= 'I/O';
		6:
		PV1	:= 'Säkerhetsläge';
	END_CASE;
END_IF;

//u01 Actual level 4002		Aktuell vätskenivå	
fbR4002(sIPAddr := sIPAddr, nTCPPort := nMBTCPPort, nUnitID := UINT_TO_BYTE(nUnitID), nQuantity := 1, bExecute := bRun, tTimeout := tTimeout,   
	nMBAddr 	:= 4001,
	cbLength	:= SIZEOF(wR4002),
	pDestAddr	:= ADR(wR4002));
	rActLevel := UINT_TO_REAL(WORD_TO_UINT(wR4002)) / 10.0;
	
//u02 Actual reference 4003	Aktuellt börvärde	
fbR4003(sIPAddr := sIPAddr, nTCPPort := nMBTCPPort, nUnitID := UINT_TO_BYTE(nUnitID), nQuantity := 1, bExecute := bRun, tTimeout := tTimeout,   
	nMBAddr 	:= 4002,
	cbLength	:= SIZEOF(wR4003),
	pDestAddr	:= ADR(wR4003));
	rActReference := UINT_TO_REAL(WORD_TO_UINT(wR4003)) / 10.0;
	
//u24 Actual OD	4004		Ventilöppningsgrad	
fbR4004(sIPAddr := sIPAddr, nTCPPort := nMBTCPPort, nUnitID := UINT_TO_BYTE(nUnitID), nQuantity := 1, bExecute := bRun, tTimeout := tTimeout,   
	nMBAddr 	:= 4003,
	cbLength	:= SIZEOF(wR4004),
	pDestAddr	:= ADR(wR4004));
	rActOD := UINT_TO_REAL(WORD_TO_UINT(wR4004)) / 10.0;

//u33 Actual valve position 4005 Ventilposition	
fbR4005(sIPAddr := sIPAddr, nTCPPort := nMBTCPPort, nUnitID := UINT_TO_BYTE(nUnitID), nQuantity := 1, bExecute := bRun, tTimeout := tTimeout,   
	nMBAddr 	:= 4004,
	cbLength	:= SIZEOF(wR4005),
	pDestAddr	:= ADR(wR4005));
	rActVP := UINT_TO_REAL(WORD_TO_UINT(wR4005)) / 10.0;

//Larmregister 1901
fbR1901(sIPAddr := sIPAddr, nTCPPort := nMBTCPPort, nUnitID := UINT_TO_BYTE(nUnitID), nQuantity := 1, bExecute := bRun, tTimeout := tTimeout,   
	nMBAddr 	:= 1900,
	cbLength	:= SIZEOF(wR1901),
	pDestAddr	:= ADR(wR1901));
	bAlarmHL 	:= wR1901.8;
	bAlarmLL 	:= wR1901.9;
	bAlarmOsc 	:= wR1901.10;
	bAlarmVP 	:= wR1901.14;
	FAULT 		:= wR1901.0;
	bSensorFault := wR1901.3;
	
	
//Kom.fel modbus
fbErrorTOF(IN := fbR1901.bError, PT := T#30S);
fbErrorTON(IN := fbErrorTOF.Q, PT := T#120S, Q => AL8);

END_FUNCTION_BLOCK

// oaksModbusLibrary/Datahantering/FB_SETPOINT_INT_MODBUS
FUNCTION_BLOCK FB_SETPOINT_INT_MODBUS
VAR_INPUT
	bPrioritySlave			: BOOL	:=TRUE;
	bSuccessModbusSlave		: BOOL;
	nActSetpointSlave		: INT;
	bValidPLCMaster			: BOOL;
	tMaxTime				: TIME	:=T#30S; 					
END_VAR

VAR_IN_OUT
	nSetpointPLCMaster		: INT;
END_VAR

VAR_OUTPUT
	nSetpointValid			: INT;
	nSetpointToSlave		: WORD;
	bSetpointUpdateSlave	: BOOL;
END_VAR

VAR
	nMemorySetpoint			: INT;
	nSeq					: INT;
	fbTimerMax				: TON;
END_VAR


fbTimerMax();

CASE nSeq OF
	0: (* Start up case first time, after power failure and max time elapsed *)
		IF bPrioritySlave AND bSuccessModbusSlave THEN
			nSetpointPLCMaster:= nActSetpointSlave;
			nMemorySetpoint:= nActSetpointSlave;
			nSetpointValid:= nActSetpointSlave;
			nSetPointToSlave:=F_INT_TO_WORD(nSetPointValid);
			bSetpointUpdateSlave:= FALSE;
			nSeq :=10;
		END_IF

		
	10: (* Control of setpoint change *)
		IF bSuccessModbusSlave AND nMemorySetpoint <> nActSetpointSlave THEN
			nSeq :=20;
		ELSIF bSuccessModbusSlave AND nMemorySetpoint <> nSetpointPLCMaster THEN
			nSeq :=30;
		END_IF

		
	20: (* Slave changed setpoint *)
			nSetpointPLCMaster:= nActSetpointSlave;
			nMemorySetpoint:= nActSetpointSlave;
			nSetpointValid:= nActSetpointSlave;
			nSetPointToSlave:=F_INT_TO_WORD(nSetPointValid);
			bSetpointUpdateSlave:= FALSE;
			nSeq :=10;

	
	30: (* PLC Master changed setpoint *)
			nMemorySetpoint:= nSetpointPLCMaster;
			nSetpointValid:= nSetpointPLCMaster;
			nSetPointToSlave:=F_INT_TO_WORD(nSetPointValid);		
			bSetpointUpdateSlave:= TRUE;
			nSeq :=31;

			
	31: (* Waiting for slave to change setpoint *)
			fbTimerMax(IN:=bSetpointUpdateSlave , PT:= tMaxTime, Q=> , ET=> );
		IF nMemorySetpoint = nActSetpointSlave THEN
			bSetpointUpdateSlave:= FALSE;
			nSeq :=10;
		ELSIF fbTimerMax.Q THEN
			bSetpointUpdateSlave:=FALSE;
			fbTimerMax();
			nSeq:=0;
		END_IF;

	
END_CASE

END_FUNCTION_BLOCK

// oaksModbusLibrary/Datahantering/fbReadGeneralModbusReg
//OAKS AB
//2022-06-22
//Funktionsblock för läsning av modbusregister funktionskod 1-4. Möjlighet för aktivering av 32bits register med litte/big endian.
//Möjlighet till 32bits läsning med swap.  
FUNCTION_BLOCK fbReadGeneralModbusReg

VAR_INPUT
	bExecute : BOOL; //Aktivering block
	sIPAddr : STRING := ''; //Ip-adress
	nTCPPort : UINT := 502; //Port
	nUnitID : BYTE := 1; //Modbus-ID
	mBusAdr : UINT; //Modbus-adress att läsa
	modbusFunction : E_Modbus_Functions_Read; 
	bRead32bit : BOOL :=FALSE; //Läs 32-bit
	bSwap : BOOL :=FALSE; //Bitordning
	tTimeout : TIME := t#5s;
END_VAR

VAR_OUTPUT
	bRead : BOOL := FALSE; //Bool-värde
	rRead : REAL := 0; //Real-värde
	bBusy : BOOL := FALSE; //Busy
	bError : BOOL := FALSE;
END_VAR

VAR
	FB_MBReadCoils_Read: FB_MBReadCoils;
	FB_MBReadInputs_Read: FB_MBReadInputs;
	FB_MBReadRegs_Read: FB_MBReadRegs;
	FB_MBReadInputRegs_Read: FB_MBReadInputRegs;
	nAddQuantity: WORD := 0;
	wRead : WORD := 0;
	R_TRIG_One: R_TRIG;
	aWordArrayNoSwap: ARRAY[0..1] OF WORD;
	aWordArrayRead: ARRAY[0..1] OF WORD;
END_VAR

R_TRIG_One(CLK:= bExecute, Q=> bRead);

IF bRead32bit THEN
	nAddQuantity := 1;
ELSE
	nAddQuantity := 0;
END_IF

CASE modbusFunction OF

	1: //Read coils 
			
		FB_MBReadCoils_Read(
		sIPAddr:= sIPAddr, 
		nTCPPort:= nTCPPort, 
		nUnitID:= nUnitID, 
		nQuantity:= 1, 
		nMBAddr:= mBusAdr, 
		cbLength:= SIZEOF(wRead), 
		pDestAddr:= ADR(WRead), 
		bExecute:= bRead, 
		tTimeout:= tTimeout, 
		bBusy=> , 
		bError=> , 
		nErrId=> , 
		cbRead=> );
		
		//Error 
		IF FB_MBReadCoils_Read.bError THEN
			FB_MBReadCoils_Read(bExecute := FALSE);
			bRead := FALSE;
			bError := TRUE;
		END_IF
		
		//Success
		IF NOT FB_MBReadCoils_Read.bBusy AND NOT FB_MBReadCoils_Read.bError THEN
			FB_MBReadCoils_Read(bExecute := FALSE);
			bRead := FALSE;
			bError := FALSE;
		END_IF	
	
		bRead := WORD_TO_BOOL(wRead);
		
	2: //Read discrete inputs
	
		FB_MBReadInputs_Read(
		sIPAddr:= sIPAddr, 
		nTCPPort:= nTCPPort, 
		nUnitID:= nUnitID, 
		nQuantity:= 1, 
		nMBAddr:= mBusAdr, 
		cbLength:= SIZEOF(wRead), 
		pDestAddr:= ADR(wRead), 
		bExecute:= bRead, 
		tTimeout:= tTimeout, 
		bBusy=> , 
		bError=> , 
		nErrId=> , 
		cbRead=> );
		
		//Error 
		IF FB_MBReadInputs_Read.bError THEN
			bRead := FALSE;
			bError := TRUE;
		END_IF
		
